C03625=1058.600,403.562,-118.922,174.891,38.797,157.435
C03626=1058.591,403.315,-118.879,174.884,38.789,157.432
C03627=1058.583,403.069,-118.835,174.877,38.781,157.430
C03628=1058.575,402.823,-118.792,174.870,38.773,157.428
C03629=1058.566,402.577,-118.749,174.863,38.765,157.426
C03630=1058.556,402.249,-118.691,174.854,38.754,157.423
C03631=1058.545,401.921,-118.634,174.845,38.744,157.420
C03632=1058.534,401.593,-118.577,174.836,38.733,157.417
C03633=1058.523,401.265,-118.519,174.828,38.723,157.414
C03634=1058.515,401.019,-118.477,174.821,38.715,157.412
C03635=1058.506,400.773,-118.434,174.814,38.707,157.410
C03636=1058.498,400.527,-118.391,174.807,38.699,157.408
C03637=1058.489,400.280,-118.348,174.800,38.691,157.406
C03638=1058.483,400.034,-118.305,174.794,38.684,157.404
C03639=1058.474,399.788,-118.262,174.787,38.676,157.402
C03640=1058.466,399.542,-118.219,174.781,38.668,157.400
C03641=1058.457,399.295,-118.177,174.774,38.660,157.398
C03642=1058.449,399.050,-118.134,174.768,38.652,157.395
C03643=1058.441,398.803,-118.092,174.761,38.644,157.393
C03644=1058.433,398.557,-118.049,174.754,38.637,157.391
C03645=1058.426,398.311,-118.006,174.748,38.629,157.389
C03646=1058.417,398.065,-117.963,174.742,38.622,157.387
C03647=1058.409,397.818,-117.921,174.735,38.614,157.385
C03648=1058.401,397.573,-117.878,174.729,38.606,157.383
C03649=1058.393,397.326,-117.836,174.722,38.599,157.381
C03650=1058.385,397.080,-117.794,174.716,38.591,157.379
C03651=1058.377,396.834,-117.751,174.710,38.583,157.377
C03652=1058.369,396.588,-117.709,174.703,38.576,157.375
C03653=1058.361,396.342,-117.667,174.696,38.568,157.373
C03654=1058.353,396.095,-117.624,174.691,38.561,157.371
C03655=1058.345,395.848,-117.582,174.684,38.554,157.369
C03656=1058.337,395.603,-117.539,174.677,38.546,157.367
C03657=1058.329,395.357,-117.497,174.672,38.539,157.365
C03658=1058.320,395.111,-117.456,174.665,38.531,157.363
C03659=1058.313,394.865,-117.414,174.659,38.524,157.361
C03660=1058.305,394.618,-117.371,174.652,38.516,157.359
C03661=1058.297,394.372,-117.330,174.647,38.509,157.357
C03662=1058.289,394.125,-117.287,174.640,38.502,157.355
C03663=1058.281,393.879,-117.245,174.633,38.494,157.353
C03664=1058.273,393.633,-117.203,174.628,38.487,157.351
C03665=1058.265,393.387,-117.161,174.621,38.479,157.349
C03666=1058.258,393.141,-117.119,174.615,38.472,157.348
C03667=1058.249,392.894,-117.078,174.609,38.465,157.346
C03668=1058.242,392.648,-117.036,174.603,38.458,157.344
C03669=1058.234,392.402,-116.994,174.597,38.451,157.342
C03670=1058.226,392.155,-116.952,174.591,38.444,157.340
C03671=1058.218,391.909,-116.911,174.584,38.436,157.338
C03672=1058.210,391.663,-116.869,174.579,38.429,157.336
C03673=1058.202,391.416,-116.827,174.572,38.422,157.334
C03674=1058.194,391.170,-116.786,174.566,38.415,157.332
C03675=1058.186,390.924,-116.744,174.560,38.408,157.330
C03676=1058.179,390.677,-116.703,174.554,38.400,157.328
C03677=1058.171,390.431,-116.661,174.548,38.393,157.327
C03678=1058.163,390.184,-116.620,174.542,38.386,157.325
C03679=1058.155,389.938,-116.578,174.537,38.379,157.323
C03680=1058.147,389.692,-116.538,174.530,38.372,157.321
C03681=1058.140,389.446,-116.496,174.525,38.365,157.319
C03682=1058.131,389.199,-116.455,174.518,38.359,157.318
C03683=1058.124,388.953,-116.413,174.512,38.352,157.316
C03684=1058.116,388.706,-116.373,174.506,38.345,157.314
C03685=1058.108,388.460,-116.331,174.500,38.338,157.312
C03686=1058.098,388.150,-116.280,174.493,38.329,157.310
C03687=1058.088,387.839,-116.228,174.486,38.320,157.308
C03688=1058.079,387.528,-116.176,174.478,38.312,157.305
C03689=1058.069,387.217,-116.124,174.471,38.303,157.303
C03690=1058.061,386.971,-116.082,174.464,38.296,157.301
C03691=1058.053,386.725,-116.042,174.459,38.289,157.299
C03692=1058.045,386.479,-116.001,174.453,38.283,157.298
C03693=1058.038,386.232,-115.960,174.447,38.276,157.296
C03694=1058.030,385.986,-115.919,174.441,38.269,157.294
C03695=1058.022,385.739,-115.878,174.436,38.262,157.292
C03696=1058.014,385.492,-115.837,174.431,38.255,157.291
C03697=1058.007,385.246,-115.798,174.424,38.249,157.289
C03698=1057.999,385.000,-115.756,174.419,38.242,157.287
C03699=1057.991,384.753,-115.716,174.413,38.235,157.285
C03700=1057.984,384.507,-115.674,174.407,38.229,157.284
C03701=1057.976,384.260,-115.634,174.401,38.222,157.282
C03702=1057.968,384.014,-115.593,174.396,38.215,157.280
C03703=1057.961,383.767,-115.553,174.391,38.209,157.279
C03704=1057.953,383.521,-115.512,174.384,38.202,157.277
C03705=1057.946,383.274,-115.471,174.379,38.196,157.275
C03706=1057.938,383.027,-115.431,174.373,38.189,157.273
C03707=1057.930,382.781,-115.390,174.368,38.183,157.272
C03708=1057.923,382.535,-115.349,174.362,38.176,157.270
C03709=1057.915,382.288,-115.309,174.356,38.169,157.268
C03710=1057.907,382.042,-115.269,174.351,38.163,157.267
C03711=1057.900,381.795,-115.228,174.345,38.156,157.265
C03712=1057.892,381.548,-115.188,174.340,38.150,157.263
C03713=1057.885,381.302,-115.148,174.334,38.143,157.262
C03714=1057.878,381.056,-115.107,174.328,38.137,157.260
C03715=1057.870,380.809,-115.067,174.323,38.130,157.258
C03716=1057.862,380.562,-115.026,174.318,38.124,157.257
C03717=1057.856,380.316,-114.986,174.312,38.117,157.255
C03718=1057.848,380.069,-114.946,174.307,38.111,157.253
C03719=1057.840,379.823,-114.906,174.301,38.105,157.252
C03720=1057.832,379.576,-114.866,174.295,38.098,157.250
C03721=1057.825,379.329,-114.826,174.290,38.092,157.248
C03722=1057.818,379.083,-114.786,174.285,38.086,157.247
C03723=1057.810,378.836,-114.746,174.279,38.079,157.245
C03724=1057.802,378.589,-114.706,174.274,38.073,157.244
C03725=1057.795,378.343,-114.666,174.269,38.067,157.242
C03726=1057.787,378.096,-114.626,174.263,38.060,157.240
C03727=1057.779,377.849,-114.586,174.257,38.054,157.239
C03728=1057.772,377.603,-114.547,174.252,38.048,157.237
C03729=1057.764,377.356,-114.507,174.247,38.042,157.236
C03730=1057.757,377.109,-114.467,174.241,38.035,157.234
C03731=1057.750,376.863,-114.427,174.236,38.029,157.233
C03732=1057.742,376.616,-114.387,174.231,38.023,157.231
C03733=1057.734,376.369,-114.348,174.226,38.017,157.229
C03734=1057.727,376.123,-114.308,174.220,38.011,157.228
C03735=1057.719,375.876,-114.268,174.215,38.004,157.226
C03736=1057.713,375.629,-114.229,174.210,37.998,157.225
C03737=1057.705,375.383,-114.189,174.205,37.992,157.223
C03738=1057.698,375.136,-114.150,174.199,37.986,157.221
C03739=1057.690,374.889,-114.110,174.194,37.980,157.220
C03740=1057.683,374.643,-114.070,174.189,37.974,157.218
C03741=1057.675,374.396,-114.031,174.184,37.968,157.217
C03742=1057.667,374.117,-113.986,174.177,37.961,157.215
C03743=1057.659,373.838,-113.942,174.171,37.954,157.213
C03744=1057.650,373.559,-113.898,174.166,37.947,157.212
C03745=1057.642,373.279,-113.853,174.159,37.940,157.210
C03746=1057.635,373.033,-113.813,174.154,37.934,157.208
C03747=1057.627,372.786,-113.773,174.149,37.928,157.207
C03748=1057.621,372.539,-113.735,174.145,37.922,157.205
C03749=1057.613,372.292,-113.695,174.139,37.916,157.204
C03750=1057.606,372.045,-113.656,174.134,37.910,157.202
C03751=1057.598,371.799,-113.617,174.129,37.905,157.201
C03752=1057.591,371.552,-113.578,174.124,37.899,157.199
C03753=1057.584,371.305,-113.539,174.119,37.893,157.198
C03754=1057.575,371.059,-113.500,174.114,37.887,157.196
C03755=1057.569,370.812,-113.461,174.108,37.881,157.195
C03756=1057.561,370.564,-113.421,174.103,37.875,157.194
C03757=1057.553,370.318,-113.383,174.098,37.869,157.192
C03758=1057.547,370.072,-113.344,174.093,37.863,157.191
C03759=1057.539,369.824,-113.304,174.088,37.858,157.189
C03760=1057.532,369.577,-113.266,174.083,37.852,157.188
C03761=1057.525,369.331,-113.227,174.078,37.846,157.186
C03762=1057.516,369.084,-113.188,174.073,37.840,157.185
C03763=1057.510,368.837,-113.149,174.067,37.834,157.183
C03764=1057.503,368.590,-113.110,174.063,37.829,157.182
C03765=1057.495,368.343,-113.072,174.058,37.823,157.180
C03766=1057.488,368.096,-113.033,174.053,37.817,157.179
C03767=1057.480,367.850,-112.995,174.048,37.811,157.178
C03768=1057.473,367.603,-112.956,174.043,37.806,157.176
C03769=1057.466,367.355,-112.917,174.038,37.800,157.175
C03770=1057.458,367.109,-112.878,174.033,37.794,157.173
C03771=1057.452,366.862,-112.840,174.029,37.789,157.172
C03772=1057.444,366.616,-112.801,174.023,37.783,157.170
C03773=1057.437,366.369,-112.763,174.018,37.777,157.169
C03774=1057.430,366.122,-112.724,174.013,37.772,157.168
C03775=1057.423,365.874,-112.686,174.008,37.766,157.166
C03776=1057.416,365.627,-112.647,174.003,37.760,157.165
C03777=1057.408,365.381,-112.609,173.999,37.755,157.163
C03778=1057.401,365.134,-112.570,173.994,37.749,157.162
C03779=1057.394,364.887,-112.532,173.989,37.743,157.161
C03780=1057.387,364.640,-112.494,173.984,37.738,157.159
C03781=1057.381,364.393,-112.455,173.979,37.732,157.158
C03782=1057.373,364.147,-112.416,173.975,37.727,157.157
C03783=1057.366,363.900,-112.378,173.970,37.721,157.155
C03784=1057.359,363.653,-112.340,173.965,37.715,157.154
C03785=1057.351,363.406,-112.301,173.960,37.710,157.152
C03786=1057.344,363.158,-112.263,173.956,37.704,157.151
C03787=1057.337,362.912,-112.225,173.951,37.699,157.150
C03788=1057.330,362.664,-112.188,173.946,37.694,157.148
C03789=1057.323,362.418,-112.149,173.941,37.688,157.147
C03790=1057.315,362.170,-112.111,173.937,37.683,157.146
C03791=1057.308,361.924,-112.073,173.932,37.677,157.144
C03792=1057.301,361.677,-112.035,173.926,37.672,157.143
C03793=1057.294,361.430,-111.997,173.921,37.666,157.142
C03794=1057.287,361.183,-111.959,173.917,37.661,157.140
C03795=1057.279,360.936,-111.922,173.912,37.655,157.139
C03796=1057.273,360.689,-111.883,173.907,37.650,157.138
C03797=1057.265,360.442,-111.845,173.902,37.645,157.136
C03798=1057.257,360.181,-111.806,173.898,37.639,157.135
C03799=1057.250,359.921,-111.765,173.893,37.633,157.133
C03800=1057.242,359.660,-111.726,173.888,37.627,157.132
C03801=1057.235,359.399,-111.686,173.883,37.622,157.131
C03802=1057.228,359.152,-111.648,173.878,37.616,157.129
C03803=1057.220,358.905,-111.610,173.873,37.611,157.128
C03804=1057.214,358.658,-111.572,173.869,37.606,157.127
C03805=1057.207,358.411,-111.534,173.864,37.600,157.125
C03806=1057.200,358.164,-111.497,173.860,37.595,157.124
C03807=1057.193,357.917,-111.459,173.855,37.590,157.123
C03808=1057.185,357.670,-111.422,173.851,37.585,157.122
C03809=1057.178,357.423,-111.384,173.847,37.579,157.120
C03810=1057.171,357.176,-111.347,173.842,37.574,157.119
C03811=1057.164,356.928,-111.309,173.837,37.569,157.118
C03812=1057.157,356.682,-111.272,173.833,37.564,157.117
C03813=1057.151,356.435,-111.234,173.828,37.558,157.115
C03814=1057.143,356.187,-111.197,173.823,37.553,157.114
C03815=1057.136,355.940,-111.159,173.819,37.548,157.113
C03816=1057.129,355.693,-111.121,173.814,37.543,157.111
C03817=1057.122,355.445,-111.085,173.809,37.538,157.110
C03818=1057.115,355.199,-111.047,173.805,37.533,157.109
C03819=1057.108,354.952,-111.010,173.800,37.527,157.108
C03820=1057.101,354.705,-110.972,173.796,37.522,157.106
C03821=1057.094,354.458,-110.935,173.791,37.517,157.105
C03822=1057.087,354.210,-110.898,173.786,37.512,157.104
C03823=1057.080,353.963,-110.861,173.782,37.507,157.103
C03824=1057.073,353.716,-110.823,173.778,37.502,157.101
C03825=1057.066,353.468,-110.787,173.774,37.497,157.100
C03826=1057.059,353.222,-110.749,173.769,37.492,157.099
C03827=1057.052,352.975,-110.712,173.765,37.486,157.098
C03828=1057.045,352.727,-110.675,173.760,37.481,157.096
C03829=1057.038,352.481,-110.638,173.756,37.476,157.095
C03830=1057.031,352.233,-110.601,173.751,37.471,157.094
C03831=1057.023,351.986,-110.564,173.746,37.466,157.093
C03832=1057.017,351.740,-110.527,173.742,37.461,157.092
C03833=1057.010,351.492,-110.490,173.738,37.456,157.090
C03834=1057.003,351.245,-110.453,173.734,37.451,157.089
C03835=1056.996,350.998,-110.416,173.729,37.446,157.088
C03836=1056.989,350.750,-110.379,173.725,37.441,157.087
C03837=1056.983,350.504,-110.342,173.720,37.436,157.086
C03838=1056.975,350.256,-110.306,173.716,37.431,157.084
C03839=1056.968,350.008,-110.269,173.711,37.426,157.083
C03840=1056.961,349.762,-110.232,173.707,37.421,157.082
C03841=1056.954,349.514,-110.195,173.703,37.416,157.081
C03842=1056.947,349.267,-110.159,173.699,37.411,157.080
C03843=1056.940,349.020,-110.122,173.694,37.406,157.078
C03844=1056.933,348.772,-110.085,173.690,37.401,157.077
C03845=1056.926,348.526,-110.049,173.685,37.397,157.076
C03846=1056.919,348.278,-110.012,173.681,37.392,157.075
C03847=1056.913,348.032,-109.975,173.676,37.387,157.074
C03848=1056.906,347.784,-109.938,173.673,37.382,157.072
C03849=1056.899,347.537,-109.903,173.668,37.377,157.071
C03850=1056.892,347.289,-109.866,173.664,37.372,157.070
C03851=1056.885,347.042,-109.829,173.660,37.367,157.069
C03852=1056.878,346.795,-109.793,173.655,37.362,157.068
C03853=1056.871,346.548,-109.757,173.651,37.358,157.067
C03854=1056.864,346.292,-109.719,173.647,37.353,157.066
C03855=1056.857,346.035,-109.681,173.643,37.348,157.064
C03856=1056.850,345.780,-109.643,173.638,37.343,157.063
C03857=1056.843,345.524,-109.605,173.633,37.338,157.062
C03858=1056.836,345.277,-109.570,173.629,37.333,157.061
C03859=1056.829,345.029,-109.533,173.625,37.327,157.060
C03860=1056.823,344.782,-109.497,173.621,37.323,157.058
C03861=1056.815,344.535,-109.461,173.617,37.318,157.057
C03862=1056.809,344.288,-109.424,173.612,37.314,157.056
C03863=1056.802,344.041,-109.388,173.608,37.308,157.055
C03864=1056.795,343.793,-109.352,173.604,37.304,157.054
C03865=1056.788,343.546,-109.315,173.600,37.299,157.053
C03866=1056.781,343.298,-109.280,173.596,37.295,157.052
C03867=1056.775,343.051,-109.243,173.592,37.289,157.050
C03868=1056.767,342.804,-109.207,173.587,37.285,157.049
C03869=1056.761,342.557,-109.171,173.583,37.280,157.048
C03870=1056.754,342.309,-109.135,173.579,37.275,157.047
C03871=1056.747,342.062,-109.100,173.575,37.271,157.046
C03872=1056.740,341.815,-109.063,173.571,37.266,157.045
C03873=1056.733,341.567,-109.028,173.566,37.261,157.044
C03874=1056.726,341.321,-108.992,173.562,37.257,157.043
C03875=1056.719,341.072,-108.956,173.559,37.252,157.042
C03876=1056.712,340.826,-108.920,173.554,37.247,157.040
C03877=1056.706,340.578,-108.883,173.550,37.243,157.039
C03878=1056.698,340.330,-108.848,173.546,37.238,157.038
C03879=1056.691,340.084,-108.812,173.542,37.233,157.037
C03880=1056.685,339.836,-108.776,173.538,37.229,157.036
C03881=1056.678,339.589,-108.740,173.534,37.224,157.035
C03882=1056.671,339.341,-108.705,173.529,37.219,157.034
C03883=1056.665,339.093,-108.669,173.526,37.215,157.033
C03884=1056.658,338.847,-108.633,173.522,37.210,157.032
C03885=1056.651,338.599,-108.598,173.517,37.206,157.031
C03886=1056.644,338.352,-108.561,173.513,37.201,157.030
C03887=1056.637,338.104,-108.526,173.510,37.197,157.029
C03888=1056.631,337.857,-108.491,173.506,37.192,157.027
C03889=1056.624,337.610,-108.455,173.501,37.187,157.026
C03890=1056.617,337.362,-108.420,173.497,37.183,157.025
C03891=1056.611,337.115,-108.384,173.494,37.178,157.024
C03892=1056.604,336.868,-108.349,173.489,37.174,157.023
C03893=1056.597,336.620,-108.312,173.485,37.169,157.022
C03894=1056.590,336.373,-108.277,173.481,37.165,157.021
C03895=1056.583,336.125,-108.242,173.478,37.160,157.020
C03896=1056.577,335.878,-108.207,173.473,37.156,157.019
C03897=1056.570,335.631,-108.172,173.469,37.151,157.018
C03898=1056.563,335.384,-108.136,173.465,37.147,157.017
C03899=1056.555,335.136,-108.101,173.462,37.142,157.016
C03900=1056.549,334.888,-108.065,173.457,37.138,157.015
C03901=1056.543,334.641,-108.030,173.453,37.133,157.014
C03902=1056.536,334.393,-107.995,173.450,37.129,157.013
C03903=1056.529,334.146,-107.959,173.446,37.124,157.011
C03904=1056.522,333.899,-107.924,173.442,37.120,157.010
C03905=1056.516,333.651,-107.889,173.437,37.115,157.009
C03906=1056.509,333.404,-107.854,173.434,37.111,157.008
C03907=1056.502,333.156,-107.819,173.430,37.107,157.007
C03908=1056.495,332.909,-107.784,173.426,37.102,157.006
C03909=1056.489,332.662,-107.749,173.422,37.098,157.005
C03910=1056.482,332.401,-107.712,173.418,37.093,157.004
C03911=1056.475,332.141,-107.675,173.414,37.088,157.003
C03912=1056.468,331.881,-107.638,173.409,37.084,157.002
C03913=1056.461,331.621,-107.601,173.406,37.079,157.001
C03914=1056.454,331.373,-107.566,173.402,37.075,157.000
C03915=1056.447,331.126,-107.531,173.398,37.070,156.999
C03916=1056.441,330.878,-107.496,173.395,37.066,156.998
C03917=1056.434,330.630,-107.461,173.390,37.062,156.997
C03918=1056.427,330.383,-107.426,173.386,37.057,156.996
C03919=1056.420,330.136,-107.391,173.383,37.053,156.995
C03920=1056.413,329.888,-107.357,173.379,37.049,156.994
C03921=1056.406,329.641,-107.322,173.375,37.044,156.993
C03922=1056.400,329.393,-107.287,173.372,37.040,156.992
C03923=1056.392,329.146,-107.253,173.367,37.036,156.991
C03924=1056.386,328.898,-107.218,173.363,37.032,156.990
C03925=1056.379,328.650,-107.183,173.360,37.027,156.989
C03926=1056.372,328.403,-107.149,173.356,37.023,156.988
C03927=1056.365,328.155,-107.114,173.352,37.019,156.987
C03928=1056.359,327.909,-107.080,173.349,37.015,156.986
C03929=1056.352,327.661,-107.046,173.344,37.010,156.985
C03930=1056.345,327.414,-107.011,173.340,37.006,156.984
C03931=1056.339,327.166,-106.976,173.337,37.002,156.983
C03932=1056.331,326.919,-106.942,173.333,36.998,156.982
C03933=1056.325,326.671,-106.907,173.329,36.993,156.981
C03934=1056.318,326.423,-106.872,173.326,36.989,156.980
C03935=1056.311,326.176,-106.838,173.322,36.985,156.979
C03936=1056.304,325.928,-106.804,173.318,36.981,156.978
C03937=1056.297,325.681,-106.769,173.315,36.977,156.977
C03938=1056.291,325.433,-106.735,173.310,36.972,156.976
C03939=1056.284,325.185,-106.701,173.307,36.968,156.975
C03940=1056.277,324.938,-106.666,173.303,36.964,156.974
C03941=1056.270,324.690,-106.632,173.299,36.960,156.973
C03942=1056.264,324.442,-106.597,173.296,36.956,156.972
C03943=1056.257,324.196,-106.563,173.292,36.951,156.971
C03944=1056.251,323.948,-106.529,173.288,36.947,156.970
C03945=1056.243,323.700,-106.495,173.285,36.943,156.969
C03946=1056.237,323.452,-106.461,173.281,36.939,156.968
C03947=1056.231,323.206,-106.426,173.277,36.935,156.968
C03948=1056.224,322.958,-106.392,173.274,36.931,156.967
C03949=1056.217,322.710,-106.358,173.270,36.926,156.966
C03950=1056.210,322.462,-106.324,173.267,36.922,156.965
C03951=1056.204,322.215,-106.290,173.263,36.918,156.964
C03952=1056.197,321.967,-106.256,173.259,36.913,156.963
C03953=1056.190,321.719,-106.221,173.256,36.909,156.962
C03954=1056.184,321.472,-106.187,173.252,36.906,156.961
C03955=1056.177,321.224,-106.154,173.248,36.901,156.960
C03956=1056.170,320.977,-106.118,173.244,36.897,156.959
C03957=1056.164,320.730,-106.085,173.240,36.893,156.958
C03958=1056.157,320.482,-106.051,173.237,36.889,156.957
C03959=1056.150,320.234,-106.017,173.233,36.884,156.956
C03960=1056.144,319.987,-105.983,173.229,36.880,156.955
C03961=1056.137,319.739,-105.949,173.226,36.876,156.954
C03962=1056.131,319.491,-105.914,173.223,36.872,156.953
C03963=1056.125,319.243,-105.881,173.219,36.868,156.952
C03964=1056.118,318.996,-105.847,173.216,36.864,156.951
C03965=1056.112,318.749,-105.813,173.212,36.860,156.950
C03966=1056.104,318.483,-105.777,173.208,36.855,156.949
C03967=1056.098,318.218,-105.741,173.204,36.851,156.948
C03968=1056.090,317.952,-105.704,173.200,36.847,156.947
C03969=1056.084,317.686,-105.668,173.197,36.842,156.946
C03970=1056.077,317.439,-105.634,173.193,36.838,156.946
C03971=1056.071,317.191,-105.600,173.190,36.834,156.945
C03972=1056.064,316.944,-105.566,173.186,36.830,156.944
C03973=1056.058,316.696,-105.532,173.182,36.826,156.943
C03974=1056.051,316.448,-105.499,173.179,36.822,156.942
C03975=1056.045,316.201,-105.465,173.175,36.818,156.941
C03976=1056.038,315.953,-105.431,173.172,36.814,156.940
C03977=1056.032,315.706,-105.397,173.168,36.810,156.939
C03978=1056.026,315.458,-105.365,173.164,36.806,156.938
C03979=1056.019,315.210,-105.330,173.162,36.801,156.937
C03980=1056.013,314.963,-105.297,173.158,36.797,156.936
C03981=1056.007,314.715,-105.263,173.155,36.793,156.935
C03982=1056.000,314.468,-105.229,173.151,36.789,156.934
C03983=1055.994,314.220,-105.195,173.147,36.785,156.933
C03984=1055.987,313.972,-105.162,173.144,36.781,156.933
C03985=1055.981,313.725,-105.129,173.140,36.777,156.932
C03986=1055.975,313.477,-105.095,173.137,36.773,156.931
C03987=1055.968,313.230,-105.062,173.133,36.769,156.930
C03988=1055.961,312.981,-105.029,173.130,36.765,156.929
C03989=1055.954,312.734,-104.995,173.126,36.761,156.928
C03990=1055.948,312.486,-104.962,173.123,36.757,156.927
C03991=1055.941,312.239,-104.929,173.120,36.753,156.926
C03992=1055.934,311.991,-104.895,173.116,36.749,156.925
C03993=1055.928,311.743,-104.863,173.113,36.745,156.925
C03994=1055.921,311.495,-104.830,173.109,36.741,156.924
C03995=1055.914,311.248,-104.796,173.106,36.737,156.923
C03996=1055.908,311.000,-104.763,173.102,36.734,156.922
C03997=1055.901,310.752,-104.730,173.099,36.730,156.921
C03998=1055.894,310.505,-104.697,173.095,36.726,156.920
C03999=1055.887,310.257,-104.664,173.091,36.722,156.919
C04000=1055.881,310.010,-104.632,173.089,36.718,156.918
C04001=1055.874,309.762,-104.599,173.085,36.714,156.918
C04002=1055.867,309.514,-104.565,173.082,36.710,156.917
C04003=1055.861,309.267,-104.532,173.078,36.706,156.916
C04004=1055.854,309.019,-104.500,173.075,36.702,156.915
C04005=1055.848,308.771,-104.466,173.071,36.699,156.914
C04006=1055.841,308.523,-104.434,173.068,36.695,156.913
C04007=1055.835,308.276,-104.401,173.065,36.691,156.912
C04008=1055.828,308.028,-104.367,173.062,36.687,156.911
C04009=1055.821,307.781,-104.335,173.058,36.683,156.911
C04010=1055.814,307.533,-104.302,173.055,36.679,156.910
C04011=1055.808,307.285,-104.269,173.051,36.675,156.909
C04012=1055.801,307.037,-104.236,173.047,36.672,156.908
C04013=1055.795,306.790,-104.204,173.044,36.668,156.907
C04014=1055.789,306.542,-104.171,173.041,36.664,156.906
C04015=1055.782,306.294,-104.138,173.038,36.660,156.905
C04016=1055.775,306.046,-104.105,173.034,36.656,156.905
C04017=1055.768,305.799,-104.073,173.031,36.652,156.904
C04018=1055.762,305.551,-104.040,173.027,36.649,156.903
C04019=1055.755,305.303,-104.007,173.025,36.645,156.902
C04020=1055.749,305.055,-103.974,173.021,36.641,156.901
C04021=1055.743,304.808,-103.942,173.018,36.637,156.900
C04022=1055.736,304.546,-103.907,173.014,36.633,156.899
C04023=1055.730,304.285,-103.873,173.011,36.629,156.898
C04024=1055.722,304.024,-103.838,173.007,36.625,156.897
C04025=1055.715,303.762,-103.804,173.003,36.621,156.897
C04026=1055.708,303.515,-103.771,173.000,36.617,156.896
C04027=1055.702,303.267,-103.739,172.997,36.613,156.895
C04028=1055.696,303.020,-103.706,172.994,36.609,156.894
C04029=1055.690,302.772,-103.674,172.990,36.606,156.893
C04030=1055.684,302.524,-103.641,172.987,36.602,156.892
C04031=1055.677,302.276,-103.609,172.984,36.598,156.892
C04032=1055.670,302.029,-103.576,172.981,36.594,156.891
C04033=1055.664,301.780,-103.544,172.977,36.590,156.890
C04034=1055.657,301.533,-103.511,172.974,36.587,156.889
C04035=1055.651,301.285,-103.478,172.971,36.583,156.888
C04036=1055.645,301.037,-103.446,172.968,36.579,156.887
C04037=1055.638,300.790,-103.414,172.964,36.575,156.886
C04038=1055.632,300.542,-103.382,172.962,36.571,156.886
C04039=1055.625,300.294,-103.349,172.958,36.568,156.885
C04040=1055.619,300.046,-103.317,172.955,36.563,156.884
C04041=1055.613,299.799,-103.284,172.951,36.559,156.883
C04042=1055.607,299.574,-103.255,172.949,36.556,156.882
C04043=1055.601,299.351,-103.226,172.945,36.552,156.881
C04044=1055.595,299.126,-103.197,172.943,36.549,156.881
C04045=1055.590,298.903,-103.168,172.940,36.546,156.880
C04046=1055.584,298.678,-103.139,172.937,36.542,156.879
C04047=1055.579,298.455,-103.110,172.934,36.539,156.879
C04048=1055.573,298.230,-103.080,172.931,36.536,156.878
C04049=1055.568,298.007,-103.050,172.929,36.532,156.877
C04050=1055.562,297.759,-103.018,172.925,36.528,156.876
C04051=1055.555,297.511,-102.987,172.923,36.524,156.875
C04052=1055.549,297.263,-102.954,172.919,36.521,156.874
C04053=1055.543,297.015,-102.922,172.916,36.517,156.874
C04054=1055.536,296.768,-102.889,172.913,36.513,156.873
C04055=1055.530,296.520,-102.858,172.910,36.509,156.872
C04056=1055.523,296.272,-102.825,172.906,36.506,156.871
C04057=1055.517,296.024,-102.794,172.904,36.502,156.870
C04058=1055.511,295.776,-102.762,172.900,36.498,156.869
C04059=1055.504,295.529,-102.730,172.897,36.495,156.869
C04060=1055.498,295.280,-102.698,172.894,36.491,156.868
C04061=1055.491,295.033,-102.666,172.891,36.487,156.867
C04062=1055.485,294.784,-102.634,172.887,36.483,156.866
C04063=1055.478,294.537,-102.602,172.885,36.479,156.865
C04064=1055.471,294.289,-102.571,172.881,36.476,156.865
C04065=1055.465,294.041,-102.539,172.878,36.472,156.864
C04066=1055.458,293.793,-102.507,172.875,36.468,156.863
C04067=1055.452,293.545,-102.474,172.872,36.465,156.862
C04068=1055.445,293.298,-102.443,172.868,36.461,156.861
C04069=1055.439,293.050,-102.412,172.866,36.457,156.861
C04070=1055.433,292.802,-102.380,172.862,36.454,156.860
C04071=1055.427,292.554,-102.348,172.859,36.450,156.859
C04072=1055.420,292.306,-102.317,172.856,36.446,156.858
C04073=1055.414,292.058,-102.285,172.853,36.443,156.857
C04074=1055.407,291.810,-102.254,172.850,36.439,156.856
C04075=1055.400,291.562,-102.222,172.847,36.435,156.856
C04076=1055.394,291.314,-102.190,172.844,36.432,156.855
C04077=1055.387,291.067,-102.158,172.841,36.428,156.854
C04078=1055.380,290.774,-102.121,172.838,36.424,156.853
C04079=1055.373,290.481,-102.084,172.834,36.419,156.852
C04080=1055.365,290.188,-102.047,172.830,36.415,156.851
C04081=1055.357,289.895,-102.009,172.826,36.410,156.850
C04082=1055.351,289.646,-101.977,172.823,36.407,156.850
C04083=1055.345,289.399,-101.946,172.820,36.403,156.849
C04084=1055.338,289.151,-101.915,172.817,36.400,156.848
C04085=1055.332,288.903,-101.883,172.814,36.396,156.847
C04086=1055.326,288.654,-101.852,172.812,36.392,156.846
C04087=1055.319,288.407,-101.821,172.808,36.389,156.846
C04088=1055.313,288.159,-101.790,172.805,36.385,156.845
C04089=1055.306,287.911,-101.758,172.802,36.381,156.844
C04090=1055.300,287.664,-101.727,172.799,36.378,156.843
C04091=1055.293,287.416,-101.695,172.796,36.374,156.842
C04092=1055.287,287.167,-101.664,172.793,36.371,156.842
C04093=1055.281,286.920,-101.633,172.790,36.367,156.841
C04094=1055.274,286.672,-101.602,172.787,36.363,156.840
C04095=1055.268,286.424,-101.570,172.783,36.360,156.839
C04096=1055.261,286.175,-101.539,172.781,36.356,156.839
C04097=1055.254,285.927,-101.508,172.778,36.353,156.838
C04098=1055.248,285.680,-101.477,172.775,36.349,156.837
C04099=1055.242,285.432,-101.446,172.772,36.346,156.836
C04100=1055.235,285.184,-101.415,172.769,36.342,156.835
C04101=1055.228,284.936,-101.383,172.766,36.338,156.835
C04102=1055.223,284.688,-101.353,172.763,36.335,156.834
C04103=1055.216,284.440,-101.322,172.760,36.331,156.833
C04104=1055.209,284.192,-101.291,172.757,36.328,156.832
C04105=1055.203,283.944,-101.260,172.754,36.324,156.832
C04106=1055.197,283.697,-101.228,172.752,36.320,156.831
C04107=1055.190,283.448,-101.198,172.748,36.316,156.830
C04108=1055.184,283.201,-101.167,172.746,36.313,156.829
C04109=1055.178,282.952,-101.136,172.742,36.309,156.828
C04110=1055.171,282.704,-101.104,172.740,36.306,156.828
C04111=1055.165,282.457,-101.074,172.736,36.302,156.827
C04112=1055.158,282.209,-101.043,172.734,36.299,156.826
C04113=1055.152,281.960,-101.012,172.730,36.295,156.825
C04114=1055.146,281.713,-100.981,172.728,36.291,156.824
C04115=1055.139,281.464,-100.950,172.725,36.288,156.824
C04116=1055.133,281.216,-100.919,172.722,36.284,156.823
C04117=1055.127,280.969,-100.888,172.719,36.281,156.822
C04118=1055.120,280.720,-100.858,172.716,36.277,156.821
C04119=1055.114,280.473,-100.827,172.713,36.273,156.821
C04120=1055.108,280.224,-100.796,172.710,36.270,156.820
C04121=1055.102,279.976,-100.765,172.707,36.266,156.819
C04122=1055.095,279.729,-100.734,172.705,36.263,156.818
C04123=1055.089,279.480,-100.703,172.701,36.259,156.818
C04124=1055.083,279.232,-100.673,172.699,36.256,156.817
C04125=1055.076,278.984,-100.642,172.695,36.252,156.816
C04126=1055.069,278.736,-100.611,172.693,36.249,156.815
C04127=1055.063,278.488,-100.581,172.691,36.245,156.815
C04128=1055.057,278.240,-100.550,172.687,36.242,156.814
C04129=1055.051,277.992,-100.520,172.685,36.238,156.813
C04130=1055.044,277.751,-100.490,172.681,36.234,156.812
C04131=1055.038,277.510,-100.460,172.679,36.231,156.812
C04132=1055.032,277.269,-100.431,172.675,36.227,156.811
C04133=1055.026,277.027,-100.400,172.673,36.224,156.810
C04134=1055.020,276.786,-100.371,172.671,36.220,156.809
C04135=1055.013,276.545,-100.342,172.667,36.217,156.809
C04136=1055.007,276.304,-100.312,172.665,36.213,156.808
C04137=1055.001,276.062,-100.282,172.662,36.210,156.807
C04138=1054.994,275.815,-100.252,172.659,36.207,156.806
C04139=1054.988,275.566,-100.221,172.657,36.203,156.806
C04140=1054.982,275.318,-100.191,172.653,36.199,156.805
C04141=1054.975,275.070,-100.161,172.651,36.196,156.804
C04142=1054.969,274.822,-100.130,172.648,36.192,156.803
C04143=1054.963,274.574,-100.100,172.645,36.189,156.803
C04144=1054.956,274.326,-100.070,172.642,36.185,156.802
C04145=1054.950,274.078,-100.039,172.639,36.182,156.801
C04146=1054.944,273.830,-100.009,172.637,36.178,156.800
C04147=1054.937,273.582,-99.979,172.634,36.175,156.800
C04148=1054.931,273.334,-99.948,172.631,36.171,156.799
C04149=1054.925,273.086,-99.918,172.628,36.168,156.798
C04150=1054.918,272.838,-99.888,172.626,36.164,156.797
C04151=1054.912,272.590,-99.858,172.623,36.161,156.797
C04152=1054.906,272.342,-99.827,172.620,36.157,156.796
C04153=1054.900,272.093,-99.798,172.617,36.153,156.795
C04154=1054.893,271.845,-99.767,172.614,36.150,156.794
C04155=1054.887,271.597,-99.737,172.612,36.146,156.794
C04156=1054.880,271.349,-99.707,172.609,36.143,156.793
C04157=1054.874,271.101,-99.677,172.606,36.139,156.792
C04158=1054.868,270.854,-99.647,172.604,36.136,156.791
C04159=1054.861,270.605,-99.617,172.600,36.133,156.791
C04160=1054.855,270.357,-99.587,172.598,36.129,156.790
C04161=1054.848,270.109,-99.557,172.595,36.126,156.789
C04162=1054.842,269.861,-99.526,172.592,36.122,156.788
C04163=1054.835,269.612,-99.497,172.590,36.119,156.788
C04164=1054.830,269.364,-99.467,172.586,36.115,156.787
C04165=1054.823,269.117,-99.437,172.584,36.112,156.786
C04166=1054.817,268.868,-99.407,172.582,36.108,156.785
C04167=1054.810,268.620,-99.377,172.578,36.105,156.785
C04168=1054.805,268.372,-99.347,172.576,36.101,156.784
C04169=1054.798,268.123,-99.317,172.573,36.098,156.783
C04170=1054.791,267.876,-99.287,172.570,36.094,156.782
C04171=1054.785,267.627,-99.257,172.568,36.090,156.782
C04172=1054.778,267.379,-99.228,172.565,36.087,156.781
C04173=1054.772,267.132,-99.198,172.562,36.083,156.780
C04174=1054.766,266.883,-99.168,172.559,36.080,156.779
C04175=1054.759,266.635,-99.138,172.557,36.076,156.779
C04176=1054.753,266.387,-99.109,172.555,36.073,156.778
C04177=1054.747,266.138,-99.078,172.551,36.070,156.777
C04178=1054.740,265.890,-99.049,172.549,36.066,156.777
C04179=1054.734,265.643,-99.020,172.546,36.063,156.776
C04180=1054.728,265.394,-98.990,172.543,36.059,156.775
C04181=1054.721,265.146,-98.960,172.541,36.056,156.774
C04182=1054.715,264.898,-98.931,172.538,36.052,156.774
C04183=1054.709,264.650,-98.901,172.535,36.049,156.773
C04184=1054.702,264.401,-98.871,172.533,36.045,156.772
C04185=1054.696,264.154,-98.841,172.530,36.041,156.771
C04186=1054.690,263.915,-98.813,172.528,36.039,156.771
C04187=1054.683,263.675,-98.784,172.525,36.035,156.770
C04188=1054.678,263.436,-98.756,172.522,36.031,156.769
C04189=1054.672,263.197,-98.728,172.520,36.028,156.768
C04190=1054.665,262.958,-98.699,172.517,36.025,156.768
C04191=1054.659,262.719,-98.670,172.515,36.021,156.767
C04192=1054.653,262.480,-98.642,172.513,36.018,156.766
C04193=1054.647,262.240,-98.613,172.509,36.015,156.766
C04194=1054.641,261.992,-98.584,172.507,36.011,156.765
C04195=1054.635,261.744,-98.555,172.504,36.008,156.764
C04196=1054.628,261.495,-98.526,172.502,36.005,156.764
C04197=1054.620,261.248,-98.497,172.499,36.001,156.763
C04198=1054.614,260.999,-98.468,172.496,35.998,156.762
C04199=1054.607,260.751,-98.438,172.494,35.994,156.761
C04200=1054.601,260.502,-98.409,172.491,35.991,156.761
C04201=1054.595,260.254,-98.380,172.488,35.988,156.760
C04202=1054.589,260.006,-98.351,172.486,35.984,156.759
C04203=1054.581,259.758,-98.321,172.483,35.981,156.759
C04204=1054.575,259.510,-98.292,172.480,35.977,156.758
C04205=1054.569,259.262,-98.263,172.478,35.974,156.757
C04206=1054.563,259.014,-98.234,172.475,35.970,156.756
C04207=1054.556,258.765,-98.205,172.473,35.967,156.756
C04208=1054.550,258.517,-98.176,172.471,35.963,156.755
C04209=1054.543,258.268,-98.146,172.467,35.960,156.754
C04210=1054.537,258.020,-98.117,172.465,35.957,156.754
C04211=1054.531,257.772,-98.088,172.463,35.953,156.753
C04212=1054.524,257.523,-98.059,172.460,35.950,156.752
C04213=1054.518,257.275,-98.030,172.457,35.946,156.751
C04214=1054.511,257.027,-98.001,172.454,35.943,156.751
C04215=1054.505,256.779,-97.972,172.452,35.940,156.750
C04216=1054.499,256.531,-97.943,172.450,35.936,156.749
C04217=1054.492,256.283,-97.914,172.447,35.933,156.749
C04218=1054.486,256.035,-97.885,172.444,35.929,156.748
C04219=1054.479,255.786,-97.856,172.442,35.925,156.747
C04220=1054.473,255.538,-97.827,172.439,35.922,156.746
C04221=1054.466,255.290,-97.798,172.437,35.919,156.746
C04222=1054.460,255.042,-97.769,172.435,35.915,156.745
C04223=1054.454,254.794,-97.740,172.432,35.912,156.744
C04224=1054.448,254.545,-97.711,172.429,35.908,156.743
C04225=1054.442,254.297,-97.682,172.426,35.905,156.743
C04226=1054.435,254.048,-97.653,172.424,35.902,156.742
C04227=1054.429,253.800,-97.624,172.422,35.898,156.741
C04228=1054.422,253.552,-97.596,172.419,35.895,156.741
C04229=1054.415,253.304,-97.566,172.417,35.891,156.740
C04230=1054.409,253.055,-97.538,172.414,35.887,156.739
C04231=1054.403,252.807,-97.509,172.411,35.884,156.738
C04232=1054.397,252.559,-97.480,172.409,35.880,156.738
C04233=1054.391,252.311,-97.451,172.407,35.877,156.737
C04234=1054.384,252.062,-97.422,172.404,35.874,156.736
C04235=1054.378,251.814,-97.394,172.402,35.870,156.736
C04236=1054.372,251.566,-97.365,172.399,35.867,156.735
C04237=1054.365,251.318,-97.336,172.396,35.863,156.734
C04238=1054.359,251.069,-97.308,172.394,35.860,156.733
C04239=1054.353,250.821,-97.279,172.391,35.856,156.733
C04240=1054.347,250.573,-97.250,172.389,35.853,156.732
C04241=1054.340,250.325,-97.221,172.387,35.849,156.731
C04242=1054.334,250.084,-97.193,172.384,35.846,156.731
C04243=1054.329,249.844,-97.165,172.382,35.842,156.730
C04244=1054.323,249.604,-97.137,172.380,35.839,156.729
C04245=1054.316,249.364,-97.110,172.377,35.836,156.728
C04246=1054.310,249.124,-97.082,172.375,35.832,156.728
C04247=1054.304,248.884,-97.055,172.373,35.829,156.727
C04248=1054.298,248.643,-97.027,172.370,35.826,156.726
C04249=1054.293,248.404,-96.999,172.368,35.822,156.726
C04250=1054.287,248.155,-96.971,172.366,35.819,156.725
C04251=1054.281,247.907,-96.942,172.363,35.815,156.724
C04252=1054.274,247.658,-96.914,172.360,35.811,156.723
C04253=1054.268,247.410,-96.885,172.357,35.808,156.723
C04254=1054.262,247.162,-96.857,172.355,35.804,156.722
C04255=1054.255,246.913,-96.828,172.353,35.801,156.721
C04256=1054.249,246.665,-96.799,172.350,35.798,156.721
C04257=1054.244,246.417,-96.771,172.348,35.794,156.720
C04258=1054.237,246.169,-96.743,172.346,35.791,156.719
C04259=1054.231,245.921,-96.714,172.343,35.787,156.718
C04260=1054.225,245.672,-96.685,172.341,35.783,156.718
C04261=1054.218,245.424,-96.658,172.339,35.780,156.717
C04262=1054.212,245.175,-96.629,172.336,35.776,156.716
C04263=1054.205,244.927,-96.601,172.334,35.773,156.716
C04264=1054.199,244.679,-96.572,172.332,35.770,156.715
C04265=1054.193,244.430,-96.544,172.329,35.766,156.714
C04266=1054.186,244.182,-96.516,172.327,35.763,156.713
C04267=1054.181,243.934,-96.487,172.325,35.759,156.713
C04268=1054.174,243.686,-96.459,172.322,35.755,156.712
C04269=1054.168,243.437,-96.431,172.319,35.752,156.711
C04270=1054.162,243.188,-96.403,172.317,35.749,156.710
C04271=1054.155,242.940,-96.374,172.314,35.745,156.710
C04272=1054.149,242.692,-96.346,172.312,35.742,156.709
C04273=1054.143,242.444,-96.319,172.310,35.738,156.708
C04274=1054.137,242.195,-96.290,172.307,35.735,156.708
C04275=1054.130,241.947,-96.262,172.305,35.731,156.707
C04276=1054.124,241.699,-96.234,172.302,35.727,156.706
C04277=1054.118,241.450,-96.206,172.300,35.724,156.705
C04278=1054.112,241.201,-96.178,172.298,35.721,156.705
C04279=1054.105,240.953,-96.150,172.295,35.717,156.704
C04280=1054.099,240.705,-96.122,172.293,35.714,156.703
C04281=1054.093,240.457,-96.093,172.291,35.711,156.703
C04282=1054.086,240.209,-96.066,172.288,35.707,156.702
C04283=1054.079,239.960,-96.038,172.286,35.704,156.701
C04284=1054.073,239.711,-96.010,172.284,35.700,156.700
C04285=1054.067,239.463,-95.982,172.281,35.696,156.700
C04286=1054.061,239.215,-95.955,172.279,35.693,156.699
C04287=1054.055,238.967,-95.926,172.277,35.690,156.698
C04288=1054.048,238.718,-95.898,172.274,35.686,156.698
C04289=1054.041,238.470,-95.871,172.272,35.683,156.697
C04290=1054.035,238.221,-95.842,172.270,35.679,156.696
C04291=1054.029,237.973,-95.815,172.268,35.676,156.696
C04292=1054.023,237.725,-95.787,172.265,35.672,156.695
C04293=1054.017,237.476,-95.759,172.263,35.669,156.694
C04294=1054.010,237.228,-95.731,172.260,35.665,156.693
C04295=1054.003,236.979,-95.704,172.258,35.662,156.693
C04296=1053.997,236.731,-95.676,172.256,35.658,156.692
C04297=1053.991,236.483,-95.648,172.254,35.655,156.691
C04298=1053.985,236.239,-95.621,172.251,35.652,156.691
C04299=1053.979,235.997,-95.595,172.249,35.648,156.690
C04300=1053.973,235.753,-95.567,172.247,35.645,156.689
C04301=1053.966,235.510,-95.539,172.245,35.641,156.688
C04302=1053.960,235.268,-95.513,172.243,35.638,156.688
C04303=1053.954,235.024,-95.486,172.241,35.634,156.687
C04304=1053.948,234.781,-95.458,172.238,35.631,156.686
C04305=1053.941,234.537,-95.431,172.236,35.628,156.686
C04306=1053.936,234.289,-95.404,172.234,35.624,156.685
C04307=1053.929,234.040,-95.376,172.231,35.620,156.684
C04308=1053.923,233.792,-95.348,172.229,35.617,156.683
C04309=1053.917,233.544,-95.321,172.227,35.613,156.683
C04310=1053.911,233.295,-95.293,172.224,35.610,156.682
C04311=1053.904,233.046,-95.266,172.222,35.607,156.681
C04312=1053.898,232.799,-95.238,172.220,35.603,156.681
C04313=1053.892,232.550,-95.211,172.217,35.600,156.680
C04314=1053.885,232.302,-95.183,172.215,35.596,156.679
C04315=1053.879,232.053,-95.156,172.214,35.592,156.679
C04316=1053.872,231.805,-95.128,172.211,35.589,156.678
C04317=1053.866,231.556,-95.100,172.209,35.586,156.677
C04318=1053.861,231.308,-95.074,172.207,35.582,156.676
C04319=1053.854,231.059,-95.046,172.204,35.579,156.676
C04320=1053.847,230.811,-95.018,172.202,35.575,156.675
C04321=1053.842,230.563,-94.991,172.200,35.571,156.674
C04322=1053.835,230.314,-94.964,172.197,35.568,156.674
C04323=1053.829,230.066,-94.936,172.195,35.564,156.673
C04324=1053.822,229.817,-94.909,172.193,35.561,156.672
C04325=1053.816,229.569,-94.882,172.190,35.558,156.671
C04326=1053.810,229.321,-94.855,172.189,35.554,156.671
C04327=1053.803,229.072,-94.827,172.187,35.550,156.670
C04328=1053.797,228.824,-94.799,172.184,35.547,156.669
C04329=1053.791,228.575,-94.773,172.182,35.543,156.669
C04330=1053.784,228.327,-94.745,172.180,35.540,156.668
C04331=1053.778,228.079,-94.718,172.178,35.537,156.667
C04332=1053.772,227.830,-94.691,172.175,35.533,156.666
C04333=1053.765,227.581,-94.664,172.173,35.529,156.666
C04334=1053.760,227.333,-94.637,172.171,35.526,156.665
C04335=1053.753,227.084,-94.609,172.169,35.523,156.664
C04336=1053.746,226.836,-94.583,172.167,35.519,156.664
C04337=1053.740,226.588,-94.556,172.165,35.516,156.663
C04338=1053.733,226.339,-94.529,172.162,35.512,156.662
C04339=1053.727,226.091,-94.501,172.160,35.508,156.662
C04340=1053.721,225.842,-94.474,172.158,35.505,156.661
C04341=1053.715,225.593,-94.447,172.155,35.502,156.660
C04342=1053.708,225.345,-94.420,172.154,35.498,156.659
C04343=1053.702,225.097,-94.394,172.152,35.495,156.659
C04344=1053.695,224.849,-94.366,172.149,35.491,156.658
C04345=1053.689,224.599,-94.339,172.147,35.487,156.657
C04346=1053.683,224.351,-94.312,172.145,35.484,156.657
C04347=1053.676,224.103,-94.285,172.143,35.480,156.656
C04348=1053.671,223.854,-94.258,172.140,35.477,156.655
C04349=1053.664,223.605,-94.231,172.139,35.474,156.654
C04350=1053.658,223.357,-94.205,172.137,35.470,156.654
C04351=1053.651,223.109,-94.177,172.134,35.466,156.653
C04352=1053.645,222.860,-94.150,172.132,35.463,156.652
C04353=1053.639,222.611,-94.123,172.130,35.459,156.652
C04354=1053.633,222.365,-94.097,172.128,35.456,156.651
C04355=1053.626,222.118,-94.071,172.126,35.452,156.650
C04356=1053.621,221.871,-94.044,172.124,35.448,156.649
C04357=1053.614,221.624,-94.017,172.121,35.445,156.649
C04358=1053.608,221.377,-93.990,172.119,35.441,156.648
C04359=1053.602,221.130,-93.963,172.118,35.438,156.647
C04360=1053.596,220.882,-93.937,172.116,35.435,156.647
C04361=1053.589,220.636,-93.910,172.113,35.431,156.646
C04362=1053.583,220.387,-93.883,172.111,35.427,156.645
C04363=1053.576,220.139,-93.857,172.109,35.424,156.644
C04364=1053.570,219.890,-93.830,172.107,35.420,156.644
C04365=1053.563,219.642,-93.803,172.105,35.417,156.643
C04366=1053.558,219.394,-93.777,172.103,35.414,156.642
C04367=1053.551,219.145,-93.750,172.100,35.410,156.642
C04368=1053.545,218.897,-93.724,172.098,35.406,156.641
C04369=1053.538,218.648,-93.697,172.097,35.403,156.640
C04370=1053.532,218.399,-93.671,172.095,35.399,156.639
C04371=1053.525,218.150,-93.644,172.092,35.396,156.639
C04372=1053.519,217.902,-93.618,172.090,35.392,156.638
C04373=1053.512,217.653,-93.591,172.088,35.388,156.637
C04374=1053.507,217.405,-93.564,172.086,35.385,156.637
C04375=1053.500,217.157,-93.538,172.084,35.382,156.636
C04376=1053.494,216.908,-93.511,172.082,35.378,156.635
C04377=1053.487,216.660,-93.485,172.079,35.374,156.635
C04378=1053.481,216.411,-93.458,172.078,35.371,156.634
C04379=1053.474,216.163,-93.432,172.076,35.367,156.633
C04380=1053.469,215.914,-93.405,172.074,35.364,156.632
C04381=1053.462,215.666,-93.379,172.071,35.360,156.632
C04382=1053.456,215.417,-93.352,172.070,35.356,156.631
C04383=1053.450,215.169,-93.325,172.068,35.353,156.630
C04384=1053.443,214.920,-93.299,172.065,35.349,156.629
C04385=1053.437,214.671,-93.273,172.063,35.346,156.629
C04386=1053.431,214.423,-93.247,172.062,35.342,156.628
C04387=1053.425,214.174,-93.220,172.059,35.338,156.627
C04388=1053.418,213.926,-93.194,172.057,35.335,156.627
C04389=1053.412,213.678,-93.167,172.055,35.331,156.626
C04390=1053.405,213.429,-93.141,172.054,35.328,156.625
C04391=1053.399,213.181,-93.114,172.051,35.324,156.624
C04392=1053.393,212.932,-93.089,172.049,35.320,156.624
C04393=1053.387,212.683,-93.062,172.048,35.317,156.623
C04394=1053.380,212.435,-93.036,172.045,35.313,156.622
C04395=1053.374,212.186,-93.009,172.043,35.309,156.622
C04396=1053.368,211.937,-92.983,172.041,35.306,156.621
C04397=1053.362,211.689,-92.957,172.040,35.303,156.620
C04398=1053.355,211.441,-92.931,172.037,35.299,156.620
C04399=1053.348,211.192,-92.904,172.035,35.296,156.619
C04400=1053.343,210.943,-92.878,172.034,35.292,156.618
C04401=1053.336,210.695,-92.852,172.031,35.288,156.617
C04402=1053.330,210.447,-92.826,172.029,35.285,156.617
C04403=1053.324,210.197,-92.800,172.027,35.281,156.616
C04404=1053.317,209.949,-92.774,172.025,35.278,156.615
C04405=1053.311,209.701,-92.748,172.023,35.274,156.614
C04406=1053.305,209.451,-92.722,172.021,35.270,156.614
C04407=1053.298,209.203,-92.696,172.020,35.267,156.613
C04408=1053.292,208.955,-92.669,172.017,35.263,156.612
C04409=1053.286,208.706,-92.644,172.015,35.259,156.612
C04410=1053.279,208.462,-92.618,172.014,35.256,156.611
C04411=1053.273,208.218,-92.593,172.011,35.252,156.610
C04412=1053.267,207.974,-92.567,172.009,35.249,156.609
C04413=1053.261,207.729,-92.541,172.008,35.245,156.609
C04414=1053.254,207.485,-92.516,172.006,35.241,156.608
C04415=1053.249,207.240,-92.491,172.003,35.238,156.607
C04416=1053.242,206.996,-92.465,172.002,35.235,156.607
C04417=1053.236,206.752,-92.440,172.000,35.231,156.606
C04418=1053.210,205.700,-92.334,171.785,35.137,156.590
C04419=1053.204,205.451,-92.309,171.783,35.135,156.589
C04420=1053.198,205.203,-92.284,171.780,35.132,156.589
C04421=1053.192,204.954,-92.259,171.777,35.129,156.588
C04422=1053.186,204.705,-92.234,171.775,35.126,156.588
C04423=1053.180,204.456,-92.209,171.773,35.124,156.587
C04424=1053.175,204.208,-92.184,171.771,35.121,156.587
C04425=1053.168,203.959,-92.159,171.768,35.118,156.586
C04426=1053.162,203.710,-92.134,171.765,35.115,156.586
C04427=1053.156,203.462,-92.110,171.763,35.113,156.585
C04428=1053.150,203.213,-92.085,171.761,35.110,156.585
C04429=1053.144,202.964,-92.060,171.758,35.107,156.584
C04430=1053.138,202.716,-92.035,171.756,35.104,156.584
C04431=1053.133,202.467,-92.011,171.753,35.102,156.583
C04432=1053.126,202.218,-91.985,171.751,35.099,156.582
C04433=1053.121,201.970,-91.961,171.748,35.096,156.582
C04434=1053.115,201.721,-91.936,171.746,35.093,156.581
C04435=1053.108,201.472,-91.912,171.744,35.091,156.581
C04436=1053.103,201.223,-91.887,171.741,35.088,156.580
C04437=1053.096,200.975,-91.863,171.738,35.085,156.580
C04438=1053.090,200.726,-91.838,171.736,35.082,156.579
C04439=1053.084,200.478,-91.813,171.734,35.080,156.579
C04440=1053.078,200.229,-91.789,171.732,35.077,156.578
C04441=1053.072,199.979,-91.764,171.728,35.074,156.578
C04442=1053.065,199.731,-91.740,171.726,35.072,156.577
C04443=1053.060,199.483,-91.715,171.724,35.069,156.577
C04444=1053.054,199.233,-91.691,171.722,35.066,156.576
C04445=1053.047,198.986,-91.666,171.719,35.064,156.576
C04446=1053.041,198.736,-91.642,171.717,35.061,156.575
C04447=1053.035,198.487,-91.618,171.714,35.058,156.575
C04448=1053.030,198.239,-91.593,171.712,35.056,156.574
C04449=1053.023,197.990,-91.569,171.709,35.053,156.574
C04450=1053.017,197.741,-91.544,171.707,35.050,156.573
C04451=1053.011,197.493,-91.520,171.705,35.048,156.573
C04452=1053.005,197.244,-91.496,171.702,35.045,156.572
C04453=1052.999,196.996,-91.471,171.699,35.042,156.572
C04454=1052.993,196.747,-91.447,171.697,35.040,156.571
C04455=1052.987,196.497,-91.422,171.695,35.037,156.571
C04456=1052.981,196.249,-91.399,171.693,35.035,156.570
C04457=1052.975,196.000,-91.374,171.691,35.032,156.570
C04458=1052.968,195.752,-91.350,171.687,35.029,156.569
C04459=1052.962,195.503,-91.325,171.685,35.027,156.569
C04460=1052.957,195.253,-91.300,171.683,35.024,156.568
C04461=1052.951,195.005,-91.277,171.681,35.021,156.568
C04462=1052.945,194.756,-91.252,171.679,35.019,156.567
C04463=1052.939,194.508,-91.228,171.676,35.016,156.567
C04464=1052.933,194.258,-91.204,171.673,35.014,156.567
C04465=1052.927,194.010,-91.180,171.671,35.011,156.566
C04466=1052.920,193.761,-91.155,171.669,35.008,156.565
C04467=1052.914,193.513,-91.131,171.667,35.006,156.565
C04468=1052.909,193.264,-91.106,171.665,35.003,156.565
C04469=1052.902,193.016,-91.083,171.661,35.000,156.564
C04470=1052.897,192.766,-91.058,171.659,34.998,156.563
C04471=1052.891,192.518,-91.034,171.657,34.995,156.563
C04472=1052.885,192.269,-91.010,171.655,34.993,156.563
C04473=1052.879,192.020,-90.986,171.653,34.990,156.562
C04474=1052.873,191.771,-90.962,171.651,34.987,156.562
C04475=1052.867,191.523,-90.938,171.647,34.985,156.561
C04476=1052.861,191.274,-90.913,171.645,34.982,156.561
C04477=1052.855,191.025,-90.890,171.643,34.980,156.560
C04478=1052.849,190.777,-90.865,171.641,34.976,156.560
C04479=1052.842,190.492,-90.838,171.639,34.974,156.559
C04480=1052.836,190.208,-90.810,171.636,34.971,156.558
C04481=1052.829,189.924,-90.783,171.633,34.968,156.558
C04482=1052.822,189.639,-90.756,171.630,34.965,156.557
C04483=1052.817,189.391,-90.732,171.628,34.962,156.557
C04484=1052.810,189.142,-90.708,171.626,34.960,156.556
C04485=1052.805,188.893,-90.683,171.624,34.957,156.556
C04486=1052.798,188.644,-90.659,171.621,34.954,156.555
C04487=1052.793,188.396,-90.635,171.619,34.952,156.555
C04488=1052.787,188.147,-90.611,171.617,34.949,156.554
C04489=1052.781,187.897,-90.588,171.614,34.947,156.554
C04490=1052.775,187.649,-90.564,171.612,34.944,156.554
C04491=1052.769,187.401,-90.540,171.610,34.941,156.553
C04492=1052.763,187.152,-90.516,171.608,34.939,156.552
C04493=1052.757,186.903,-90.492,171.605,34.936,156.552
C04494=1052.752,186.654,-90.468,171.603,34.934,156.552
C04495=1052.746,186.405,-90.444,171.601,34.931,156.551
C04496=1052.740,186.157,-90.420,171.599,34.928,156.550
C04497=1052.734,185.908,-90.396,171.597,34.926,156.550
C04498=1052.729,185.658,-90.373,171.595,34.923,156.550
C04499=1052.723,185.410,-90.349,171.591,34.921,156.549
C04500=1052.717,185.162,-90.325,171.589,34.918,156.549
C04501=1052.711,184.913,-90.301,171.587,34.916,156.548
C04502=1052.705,184.664,-90.278,171.585,34.912,156.548
C04503=1052.700,184.415,-90.253,171.583,34.910,156.547
C04504=1052.693,184.166,-90.229,171.581,34.907,156.547
C04505=1052.687,183.917,-90.206,171.578,34.905,156.546
C04506=1052.681,183.669,-90.183,171.576,34.902,156.546
C04507=1052.675,183.419,-90.159,171.574,34.900,156.545
C04508=1052.669,183.171,-90.136,171.572,34.897,156.545
C04509=1052.663,182.921,-90.113,171.569,34.896,156.544
C04510=1052.657,182.673,-90.089,171.567,34.893,156.544
C04511=1052.651,182.425,-90.065,171.565,34.891,156.544
C04512=1052.644,182.175,-90.042,171.562,34.888,156.543
C04513=1052.638,181.927,-90.018,171.560,34.886,156.543
C04514=1052.632,181.678,-89.995,171.558,34.883,156.542
C04515=1052.626,181.429,-89.972,171.556,34.881,156.542
C04516=1052.620,181.180,-89.948,171.554,34.878,156.541
C04517=1052.614,180.932,-89.926,171.552,34.876,156.541
C04518=1052.607,180.683,-89.902,171.549,34.874,156.540
C04519=1052.601,180.434,-89.879,171.547,34.871,156.540
C04520=1052.595,180.186,-89.855,171.544,34.869,156.540
C04521=1052.589,179.936,-89.832,171.542,34.866,156.539
C04522=1052.583,179.688,-89.808,171.540,34.864,156.539
C04523=1052.577,179.439,-89.785,171.538,34.861,156.538
C04524=1052.571,179.189,-89.762,171.536,34.859,156.538
C04525=1052.565,178.941,-89.738,171.533,34.857,156.537
C04526=1052.559,178.692,-89.715,171.531,34.854,156.537
C04527=1052.553,178.442,-89.692,171.529,34.852,156.536
C04528=1052.547,178.194,-89.668,171.527,34.849,156.536
C04529=1052.540,177.946,-89.646,171.525,34.847,156.536
C04530=1052.534,177.697,-89.622,171.523,34.844,156.535
C04531=1052.528,177.448,-89.599,171.521,34.842,156.535
C04532=1052.522,177.199,-89.576,171.518,34.840,156.534
C04533=1052.516,176.950,-89.553,171.516,34.837,156.534
C04534=1052.510,176.702,-89.530,171.514,34.835,156.533
C04535=1052.504,176.452,-89.506,171.512,34.832,156.533
C04536=1052.498,176.203,-89.483,171.510,34.830,156.532
C04537=1052.491,175.955,-89.460,171.508,34.827,156.532
C04538=1052.486,175.706,-89.437,171.505,34.825,156.532
C04539=1052.479,175.457,-89.414,171.502,34.823,156.531
C04540=1052.474,175.208,-89.391,171.500,34.820,156.531
C04541=1052.468,174.959,-89.367,171.498,34.818,156.530
C04542=1052.462,174.711,-89.344,171.496,34.815,156.530
C04543=1052.455,174.426,-89.319,171.494,34.813,156.529
C04544=1052.448,174.141,-89.291,171.492,34.810,156.529
C04545=1052.441,173.857,-89.266,171.489,34.807,156.528
C04546=1052.435,173.572,-89.239,171.486,34.805,156.528
C04547=1052.428,173.323,-89.215,171.484,34.802,156.527
C04548=1052.422,173.074,-89.193,171.482,34.800,156.527
C04549=1052.416,172.826,-89.170,171.480,34.797,156.526
C04550=1052.410,172.577,-89.147,171.478,34.795,156.526
C04551=1052.405,172.328,-89.124,171.476,34.792,156.526
C04552=1052.399,172.079,-89.101,171.474,34.790,156.525
C04553=1052.393,171.830,-89.078,171.471,34.788,156.525
C04554=1052.386,171.581,-89.056,171.469,34.785,156.524
C04555=1052.380,171.332,-89.033,171.467,34.783,156.524
C04556=1052.374,171.084,-89.009,171.465,34.780,156.523
C04557=1052.369,170.835,-88.986,171.463,34.778,156.523
C04558=1052.363,170.586,-88.963,171.461,34.775,156.522
C04559=1052.357,170.337,-88.940,171.459,34.773,156.522
C04560=1052.351,170.088,-88.918,171.457,34.771,156.522
C04561=1052.345,169.839,-88.895,171.454,34.768,156.521
C04562=1052.339,169.590,-88.872,171.452,34.766,156.521
C04563=1052.333,169.342,-88.849,171.450,34.763,156.520
C04564=1052.328,169.093,-88.826,171.448,34.761,156.520
C04565=1052.322,168.844,-88.803,171.446,34.759,156.519
C04566=1052.315,168.594,-88.780,171.444,34.757,156.519
C04567=1052.309,168.346,-88.757,171.442,34.754,156.519
C04568=1052.303,168.097,-88.735,171.440,34.752,156.518
C04569=1052.298,167.848,-88.712,171.438,34.749,156.518
C04570=1052.292,167.599,-88.689,171.436,34.747,156.517
C04571=1052.286,167.350,-88.667,171.434,34.745,156.517
C04572=1052.280,167.101,-88.644,171.432,34.742,156.516
C04573=1052.274,166.852,-88.621,171.430,34.740,156.516
C04574=1052.269,166.603,-88.598,171.428,34.737,156.515
C04575=1052.263,166.354,-88.575,171.425,34.735,156.515
C04576=1052.256,166.105,-88.553,171.423,34.733,156.515
C04577=1052.251,165.857,-88.530,171.421,34.730,156.514
C04578=1052.245,165.608,-88.507,171.419,34.728,156.514
C04579=1052.239,165.359,-88.484,171.417,34.725,156.513
C04580=1052.233,165.110,-88.462,171.415,34.723,156.513
C04581=1052.227,164.861,-88.439,171.413,34.720,156.512
C04582=1052.222,164.612,-88.417,171.411,34.718,156.512
C04583=1052.217,164.364,-88.394,171.408,34.716,156.512
C04584=1052.210,164.115,-88.372,171.407,34.713,156.511
C04585=1052.204,163.866,-88.349,171.405,34.711,156.511
C04586=1052.199,163.617,-88.326,171.403,34.708,156.510
C04587=1052.193,163.368,-88.303,171.401,34.706,156.510
C04588=1052.187,163.119,-88.281,171.399,34.704,156.509
C04589=1052.181,162.870,-88.258,171.397,34.701,156.509
C04590=1052.176,162.621,-88.236,171.395,34.699,156.509
C04591=1052.170,162.372,-88.213,171.392,34.696,156.508
C04592=1052.164,162.123,-88.190,171.390,34.694,156.508
C04593=1052.158,161.874,-88.168,171.388,34.691,156.507
C04594=1052.152,161.625,-88.145,171.387,34.689,156.507
C04595=1052.147,161.377,-88.123,171.385,34.687,156.506
C04596=1052.141,161.128,-88.100,171.383,34.684,156.506
C04597=1052.135,160.879,-88.078,171.381,34.682,156.505
C04598=1052.129,160.630,-88.055,171.378,34.679,156.505
C04599=1052.123,160.381,-88.033,171.376,34.677,156.505
C04600=1052.118,160.132,-88.011,171.374,34.675,156.504
C04601=1052.111,159.883,-87.988,171.372,34.673,156.504
C04602=1052.105,159.634,-87.967,171.370,34.670,156.503
C04603=1052.099,159.385,-87.944,171.368,34.668,156.503
C04604=1052.093,159.136,-87.922,171.366,34.666,156.503
C04605=1052.087,158.887,-87.899,171.365,34.664,156.502
C04606=1052.081,158.638,-87.877,171.363,34.661,156.502
C04607=1052.074,158.353,-87.852,171.359,34.659,156.501
C04608=1052.068,158.068,-87.827,171.357,34.656,156.501
C04609=1052.060,157.783,-87.801,171.355,34.653,156.500
C04610=1052.054,157.498,-87.776,171.353,34.651,156.500
C04611=1052.048,157.249,-87.753,171.351,34.648,156.499
C04612=1052.042,157.000,-87.731,171.349,34.647,156.499
C04613=1052.035,156.751,-87.709,171.347,34.644,156.499
C04614=1052.030,156.502,-87.687,171.345,34.641,156.498
C04615=1052.024,156.254,-87.665,171.343,34.640,156.498
C04616=1052.018,156.004,-87.643,171.341,34.637,156.497
C04617=1052.012,155.756,-87.620,171.339,34.635,156.497
C04618=1052.006,155.506,-87.599,171.337,34.633,156.497
C04619=1052.000,155.257,-87.577,171.335,34.630,156.496
C04620=1051.994,155.008,-87.554,171.333,34.628,156.496
C04621=1051.988,154.759,-87.532,171.331,34.626,156.495
C04622=1051.981,154.510,-87.510,171.329,34.623,156.495
C04623=1051.976,154.262,-87.489,171.327,34.621,156.495
C04624=1051.970,154.012,-87.467,171.325,34.619,156.494
C04625=1051.964,153.764,-87.444,171.323,34.617,156.494
C04626=1051.958,153.515,-87.423,171.321,34.614,156.493
C04627=1051.952,153.265,-87.401,171.319,34.612,156.493
C04628=1051.946,153.017,-87.378,171.317,34.610,156.493
C04629=1051.940,152.768,-87.357,171.315,34.608,156.492
C04630=1051.934,152.519,-87.335,171.313,34.605,156.492
C04631=1051.928,152.270,-87.313,171.312,34.603,156.491
C04632=1051.921,152.021,-87.291,171.309,34.601,156.491
C04633=1051.916,151.772,-87.269,171.307,34.599,156.490
C04634=1051.910,151.522,-87.247,171.305,34.597,156.490
C04635=1051.904,151.274,-87.225,171.303,34.594,156.490
C04636=1051.898,151.025,-87.204,171.301,34.592,156.489
C04637=1051.892,150.776,-87.182,171.299,34.590,156.489
C04638=1051.886,150.527,-87.160,171.298,34.587,156.488
C04639=1051.881,150.278,-87.138,171.296,34.585,156.488
C04640=1051.874,150.029,-87.116,171.294,34.583,156.488
C04641=1051.868,149.780,-87.094,171.291,34.581,156.487
C04642=1051.862,149.531,-87.073,171.289,34.578,156.487
C04643=1051.856,149.282,-87.051,171.287,34.576,156.487
C04644=1051.851,149.033,-87.029,171.286,34.574,156.486
C04645=1051.844,148.784,-87.007,171.284,34.572,156.486
C04646=1051.838,148.535,-86.985,171.282,34.569,156.485
C04647=1051.832,148.286,-86.964,171.280,34.568,156.485
C04648=1051.827,148.037,-86.942,171.278,34.565,156.484
C04649=1051.820,147.788,-86.921,171.276,34.562,156.484
C04650=1051.814,147.539,-86.899,171.274,34.561,156.484
C04651=1051.808,147.290,-86.878,171.272,34.558,156.483
C04652=1051.803,147.041,-86.856,171.270,34.556,156.483
C04653=1051.796,146.792,-86.835,171.268,34.554,156.483
C04654=1051.790,146.543,-86.813,171.266,34.552,156.482
C04655=1051.784,146.294,-86.791,171.264,34.550,156.482
C04656=1051.778,146.046,-86.769,171.263,34.547,156.481
C04657=1051.772,145.797,-86.748,171.261,34.545,156.481
C04658=1051.766,145.547,-86.726,171.259,34.543,156.481
C04659=1051.760,145.298,-86.704,171.257,34.541,156.480
C04660=1051.754,145.050,-86.683,171.254,34.538,156.480
C04661=1051.748,144.801,-86.662,171.252,34.536,156.479
C04662=1051.742,144.551,-86.640,171.251,34.534,156.479
C04663=1051.736,144.302,-86.618,171.249,34.532,156.479
C04664=1051.730,144.053,-86.598,171.247,34.530,156.478
C04665=1051.723,143.804,-86.577,171.245,34.528,156.478
C04666=1051.717,143.555,-86.555,171.243,34.526,156.478
C04667=1051.712,143.306,-86.534,171.242,34.523,156.477
C04668=1051.706,143.057,-86.512,171.240,34.521,156.477
C04669=1051.699,142.808,-86.491,171.238,34.519,156.476
C04670=1051.694,142.559,-86.469,171.235,34.517,156.476
C04671=1051.687,142.274,-86.444,171.233,34.514,156.475
C04672=1051.680,141.988,-86.420,171.231,34.512,156.475
C04673=1051.673,141.703,-86.395,171.229,34.509,156.475
C04674=1051.667,141.418,-86.371,171.227,34.507,156.474
C04675=1051.660,141.169,-86.350,171.225,34.504,156.474
C04676=1051.654,140.920,-86.329,171.223,34.502,156.473
C04677=1051.648,140.671,-86.307,171.222,34.500,156.473
C04678=1051.642,140.422,-86.285,171.220,34.498,156.473
C04679=1051.636,140.173,-86.264,171.217,34.495,156.472
C04680=1051.630,139.924,-86.243,171.215,34.493,156.472
C04681=1051.624,139.674,-86.222,171.213,34.491,156.471
C04682=1051.619,139.426,-86.200,171.212,34.489,156.471
C04683=1051.612,139.177,-86.179,171.210,34.487,156.471
C04684=1051.606,138.928,-86.158,171.208,34.484,156.470
C04685=1051.601,138.678,-86.137,171.206,34.483,156.470
C04686=1051.594,138.429,-86.116,171.204,34.480,156.469
C04687=1051.588,138.181,-86.095,171.203,34.478,156.469
C04688=1051.582,137.932,-86.073,171.201,34.476,156.469
C04689=1051.576,137.682,-86.052,171.198,34.474,156.468
C04690=1051.571,137.434,-86.031,171.196,34.472,156.468
C04691=1051.564,137.185,-86.010,171.195,34.469,156.467
C04692=1051.558,136.935,-85.989,171.193,34.467,156.467
C04693=1051.552,136.686,-85.968,171.191,34.465,156.467
C04694=1051.545,136.437,-85.947,171.189,34.463,156.466
C04695=1051.540,136.188,-85.926,171.187,34.461,156.466
C04696=1051.534,135.939,-85.905,171.186,34.458,156.466
C04697=1051.528,135.691,-85.883,171.184,34.457,156.465
C04698=1051.522,135.441,-85.863,171.182,34.455,156.465
C04699=1051.516,135.192,-85.841,171.180,34.452,156.464
C04700=1051.510,134.943,-85.820,171.178,34.450,156.464
C04701=1051.503,134.694,-85.800,171.176,34.448,156.464
C04702=1051.498,134.445,-85.778,171.174,34.446,156.463
C04703=1051.492,134.195,-85.758,171.172,34.444,156.463
C04704=1051.486,133.947,-85.737,171.171,34.441,156.463
C04705=1051.480,133.698,-85.715,171.169,34.439,156.462
C04706=1051.474,133.449,-85.695,171.167,34.437,156.462
C04707=1051.467,133.200,-85.674,171.165,34.435,156.461
C04708=1051.462,132.951,-85.653,171.164,34.433,156.461
C04709=1051.456,132.702,-85.631,171.162,34.430,156.461
C04710=1051.449,132.452,-85.611,171.159,34.428,156.460
C04711=1051.444,132.204,-85.590,171.157,34.426,156.460
C04712=1051.438,131.954,-85.569,171.156,34.424,156.460
C04713=1051.432,131.706,-85.548,171.154,34.422,156.459
C04714=1051.426,131.456,-85.527,171.152,34.420,156.459
C04715=1051.419,131.208,-85.507,171.150,34.418,156.458
C04716=1051.414,130.958,-85.486,171.149,34.416,156.458
C04717=1051.407,130.710,-85.465,171.147,34.413,156.458
C04718=1051.401,130.460,-85.445,171.145,34.411,156.457
C04719=1051.395,130.211,-85.424,171.143,34.409,156.457
C04720=1051.389,129.962,-85.403,171.142,34.407,156.457
C04721=1051.382,129.713,-85.383,171.139,34.405,156.456
C04722=1051.376,129.464,-85.362,171.137,34.403,156.456
C04723=1051.370,129.215,-85.341,171.135,34.401,156.456
C04724=1051.365,128.965,-85.321,171.134,34.399,156.455
C04725=1051.358,128.717,-85.300,171.132,34.397,156.455
C04726=1051.352,128.468,-85.280,171.130,34.395,156.454
C04727=1051.346,128.218,-85.259,171.128,34.393,156.454
C04728=1051.340,127.970,-85.238,171.127,34.391,156.454
C04729=1051.333,127.720,-85.218,171.125,34.388,156.453
C04730=1051.328,127.471,-85.197,171.123,34.386,156.453
C04731=1051.321,127.222,-85.176,171.121,34.384,156.453
C04732=1051.315,126.973,-85.156,171.120,34.383,156.452
C04733=1051.309,126.724,-85.135,171.117,34.380,156.452
C04734=1051.303,126.475,-85.115,171.115,34.378,156.452
C04735=1051.296,126.189,-85.092,171.113,34.376,156.451
C04736=1051.289,125.904,-85.068,171.111,34.373,156.451
C04737=1051.282,125.619,-85.044,171.109,34.371,156.450
C04738=1051.275,125.333,-85.021,171.107,34.369,156.450
C04739=1051.268,125.084,-85.000,171.105,34.367,156.450
C04740=1051.263,124.835,-84.980,171.104,34.364,156.449
C04741=1051.256,124.585,-84.960,171.102,34.362,156.449
C04742=1051.250,124.337,-84.939,171.100,34.360,156.448
C04743=1051.244,124.087,-84.918,171.099,34.358,156.448
C04744=1051.238,123.838,-84.898,171.096,34.356,156.448
C04745=1051.232,123.589,-84.878,171.094,34.354,156.447
C04746=1051.226,123.340,-84.857,171.092,34.352,156.447
C04747=1051.220,123.091,-84.836,171.091,34.349,156.447
C04748=1051.214,122.842,-84.816,171.089,34.347,156.446
C04749=1051.208,122.593,-84.796,171.087,34.345,156.446
C04750=1051.202,122.344,-84.776,171.086,34.343,156.445
C04751=1051.196,122.094,-84.755,171.084,34.341,156.445
C04752=1051.190,121.845,-84.735,171.082,34.339,156.445
C04753=1051.184,121.596,-84.714,171.080,34.337,156.444
C04754=1051.178,121.348,-84.694,171.079,34.335,156.444
C04755=1051.172,121.098,-84.673,171.077,34.333,156.444
C04756=1051.166,120.849,-84.653,171.074,34.331,156.443
C04757=1051.160,120.600,-84.633,171.073,34.328,156.443
C04758=1051.154,120.351,-84.613,171.071,34.326,156.443
C04759=1051.148,120.101,-84.592,171.069,34.324,156.442
C04760=1051.142,119.853,-84.572,171.068,34.322,156.442
C04761=1051.136,119.604,-84.552,171.066,34.320,156.441
C04762=1051.130,119.354,-84.531,171.064,34.318,156.441
C04763=1051.124,119.105,-84.511,171.062,34.315,156.441
C04764=1051.118,118.856,-84.491,171.061,34.314,156.440
C04765=1051.111,118.607,-84.471,171.059,34.312,156.440
C04766=1051.106,118.358,-84.450,171.057,34.309,156.440
C04767=1051.100,118.109,-84.430,171.056,34.307,156.439
C04768=1051.094,117.859,-84.410,171.053,34.305,156.439
C04769=1051.088,117.610,-84.389,171.051,34.303,156.438
C04770=1051.082,117.362,-84.370,171.050,34.301,156.438
C04771=1051.076,117.113,-84.350,171.048,34.299,156.438
C04772=1051.070,116.863,-84.329,171.046,34.296,156.437
C04773=1051.065,116.614,-84.309,171.045,34.294,156.437
C04774=1051.059,116.365,-84.289,171.043,34.292,156.437
C04775=1051.052,116.116,-84.268,171.041,34.290,156.436
C04776=1051.046,115.867,-84.248,171.040,34.288,156.436
C04777=1051.041,115.618,-84.228,171.038,34.286,156.436
C04778=1051.035,115.369,-84.208,171.036,34.284,156.435
C04779=1051.028,115.119,-84.188,171.035,34.282,156.435
C04780=1051.022,114.871,-84.168,171.033,34.280,156.434
C04781=1051.017,114.622,-84.147,171.030,34.277,156.434
C04782=1051.011,114.373,-84.127,171.029,34.275,156.434
C04783=1051.005,114.124,-84.107,171.027,34.273,156.433
C04784=1050.999,113.874,-84.088,171.025,34.271,156.433
C04785=1050.993,113.625,-84.068,171.024,34.269,156.433
C04786=1050.987,113.376,-84.047,171.022,34.267,156.432
C04787=1050.981,113.126,-84.027,171.020,34.265,156.432
C04788=1050.975,112.878,-84.007,171.019,34.262,156.431
C04789=1050.969,112.628,-83.988,171.017,34.260,156.431
C04790=1050.963,112.379,-83.968,171.015,34.259,156.431
C04791=1050.956,112.130,-83.947,171.014,34.257,156.430
C04792=1050.950,111.881,-83.927,171.012,34.254,156.430
C04793=1050.944,111.632,-83.907,171.010,34.252,156.430
C04794=1050.939,111.383,-83.888,171.008,34.250,156.429
C04795=1050.932,111.133,-83.868,171.006,34.248,156.429
C04796=1050.926,110.884,-83.848,171.004,34.246,156.429
C04797=1050.919,110.636,-83.828,171.003,34.244,156.428
C04798=1050.914,110.386,-83.809,171.001,34.242,156.428
C04799=1050.907,110.100,-83.786,170.999,34.239,156.427
C04800=1050.899,109.815,-83.763,170.997,34.237,156.427
C04801=1050.893,109.529,-83.740,170.995,34.235,156.427
C04802=1050.885,109.244,-83.718,170.993,34.233,156.426
C04803=1050.879,108.994,-83.699,170.991,34.230,156.426
C04804=1050.873,108.745,-83.679,170.990,34.228,156.426
C04805=1050.867,108.497,-83.659,170.988,34.226,156.425
C04806=1050.861,108.246,-83.639,170.986,34.224,156.425
C04807=1050.854,107.998,-83.620,170.984,34.223,156.425
C04808=1050.848,107.749,-83.600,170.982,34.221,156.424
C04809=1050.843,107.500,-83.581,170.980,34.218,156.424
C04810=1050.837,107.251,-83.561,170.979,34.216,156.423
C04811=1050.831,107.001,-83.541,170.977,34.214,156.423
C04812=1050.825,106.752,-83.521,170.975,34.212,156.423
C04813=1050.818,106.503,-83.502,170.974,34.210,156.422
C04814=1050.812,106.254,-83.482,170.972,34.208,156.422
C04815=1050.806,106.005,-83.462,170.970,34.206,156.422
C04816=1050.800,105.755,-83.443,170.969,34.204,156.421
C04817=1050.794,105.506,-83.423,170.967,34.202,156.421
C04818=1050.788,105.257,-83.404,170.966,34.200,156.421
C04819=1050.781,105.008,-83.384,170.964,34.198,156.420
C04820=1050.776,104.759,-83.365,170.962,34.196,156.420
C04821=1050.770,104.510,-83.345,170.960,34.194,156.420
C04822=1050.764,104.261,-83.326,170.958,34.192,156.419
C04823=1050.757,104.011,-83.306,170.956,34.190,156.419
C04824=1050.752,103.762,-83.286,170.955,34.187,156.419
C04825=1050.745,103.513,-83.267,170.953,34.185,156.418
C04826=1050.739,103.264,-83.248,170.951,34.183,156.418
C04827=1050.733,103.015,-83.228,170.950,34.181,156.418
C04828=1050.728,102.765,-83.208,170.948,34.179,156.417
C04829=1050.722,102.517,-83.189,170.946,34.177,156.417
C04830=1050.715,102.268,-83.170,170.945,34.175,156.416
C04831=1050.709,102.019,-83.150,170.943,34.173,156.416
C04832=1050.703,101.769,-83.130,170.941,34.171,156.416
C04833=1050.697,101.519,-83.111,170.940,34.169,156.415
C04834=1050.691,101.270,-83.091,170.938,34.167,156.415
C04835=1050.685,101.021,-83.072,170.936,34.165,156.415
C04836=1050.679,100.772,-83.052,170.934,34.163,156.414
C04837=1050.673,100.523,-83.033,170.932,34.161,156.414
C04838=1050.667,100.274,-83.015,170.931,34.158,156.414
C04839=1050.661,100.025,-82.995,170.929,34.156,156.413
C04840=1050.655,99.776,-82.975,170.927,34.154,156.413
C04841=1050.648,99.526,-82.956,170.926,34.153,156.413
C04842=1050.642,99.277,-82.936,170.924,34.151,156.412
C04843=1050.636,99.028,-82.918,170.922,34.149,156.412
C04844=1050.630,98.778,-82.899,170.921,34.147,156.412
C04845=1050.623,98.530,-82.879,170.919,34.145,156.411
C04846=1050.617,98.280,-82.860,170.917,34.143,156.411
C04847=1050.611,98.031,-82.841,170.916,34.140,156.410
C04848=1050.605,97.782,-82.822,170.914,34.138,156.410
C04849=1050.599,97.533,-82.802,170.912,34.136,156.410
C04850=1050.593,97.284,-82.783,170.911,34.134,156.410
C04851=1050.587,97.035,-82.764,170.908,34.132,156.409
C04852=1050.581,96.785,-82.746,170.907,34.131,156.409
C04853=1050.574,96.536,-82.725,170.905,34.129,156.409
C04854=1050.568,96.287,-82.707,170.903,34.127,156.408
C04855=1050.562,96.037,-82.687,170.902,34.124,156.408
C04856=1050.556,95.788,-82.669,170.900,34.122,156.407
C04857=1050.550,95.539,-82.649,170.898,34.120,156.407
C04858=1050.543,95.290,-82.630,170.897,34.118,156.407
C04859=1050.538,95.041,-82.611,170.895,34.116,156.406
C04860=1050.532,94.791,-82.592,170.893,34.114,156.406
C04861=1050.525,94.542,-82.573,170.892,34.113,156.406
C04862=1050.520,94.293,-82.554,170.890,34.110,156.405
C04863=1050.513,94.008,-82.532,170.888,34.108,156.405
C04864=1050.506,93.722,-82.510,170.886,34.105,156.405
C04865=1050.499,93.437,-82.488,170.885,34.103,156.404
C04866=1050.492,93.150,-82.466,170.882,34.101,156.404
C04867=1050.485,92.902,-82.447,170.880,34.099,156.404
C04868=1050.479,92.652,-82.428,170.878,34.097,156.403
C04869=1050.473,92.403,-82.409,170.877,34.095,156.403
C04870=1050.467,92.154,-82.390,170.875,34.093,156.402
C04871=1050.461,91.905,-82.371,170.874,34.091,156.402
C04872=1050.455,91.655,-82.352,170.872,34.089,156.402
C04873=1050.449,91.406,-82.333,170.870,34.087,156.401
C04874=1050.443,91.157,-82.314,170.869,34.085,156.401
C04875=1050.437,90.908,-82.296,170.867,34.083,156.401
C04876=1050.432,90.659,-82.277,170.865,34.080,156.400
C04877=1050.425,90.410,-82.258,170.864,34.078,156.400
C04878=1050.419,90.160,-82.239,170.862,34.076,156.400
C04879=1050.413,89.911,-82.220,170.861,34.074,156.399
C04880=1050.407,89.662,-82.201,170.859,34.072,156.399
C04881=1050.400,89.413,-82.183,170.857,34.071,156.399
C04882=1050.394,89.163,-82.164,170.855,34.069,156.398
C04883=1050.388,88.914,-82.145,170.853,34.067,156.398
C04884=1050.382,88.665,-82.126,170.851,34.065,156.398
C04885=1050.375,88.416,-82.108,170.850,34.063,156.397
C04886=1050.370,88.167,-82.088,170.848,34.061,156.397
C04887=1050.363,87.918,-82.070,170.846,34.059,156.397
C04888=1050.357,87.668,-82.051,170.845,34.057,156.396
C04889=1050.350,87.419,-82.032,170.843,34.055,156.396
C04890=1050.345,87.170,-82.013,170.842,34.053,156.396
C04891=1050.338,86.920,-81.995,170.840,34.051,156.395
C04892=1050.332,86.671,-81.977,170.838,34.049,156.395
C04893=1050.326,86.422,-81.958,170.837,34.047,156.395
C04894=1050.320,86.172,-81.939,170.835,34.045,156.394
C04895=1050.313,85.923,-81.920,170.833,34.043,156.394
C04896=1050.307,85.674,-81.901,170.832,34.041,156.394
C04897=1050.301,85.425,-81.883,170.830,34.039,156.393
C04898=1050.295,85.175,-81.865,170.829,34.037,156.393
C04899=1050.289,84.927,-81.846,170.827,34.035,156.393
C04900=1050.283,84.677,-81.827,170.824,34.033,156.392
C04901=1050.277,84.428,-81.809,170.823,34.031,156.392
C04902=1050.270,84.179,-81.790,170.821,34.029,156.392
C04903=1050.264,83.930,-81.771,170.819,34.027,156.391
C04904=1050.258,83.680,-81.753,170.818,34.025,156.391
C04905=1050.252,83.431,-81.734,170.816,34.023,156.391
C04906=1050.245,83.182,-81.716,170.815,34.021,156.390
C04907=1050.240,82.933,-81.697,170.813,34.019,156.390
C04908=1050.234,82.683,-81.679,170.811,34.017,156.390
C04909=1050.228,82.434,-81.660,170.810,34.015,156.389
C04910=1050.221,82.185,-81.641,170.808,34.013,156.389
C04911=1050.215,81.936,-81.623,170.806,34.011,156.389
C04912=1050.209,81.686,-81.605,170.805,34.009,156.388
C04913=1050.203,81.437,-81.586,170.803,34.007,156.388
C04914=1050.197,81.188,-81.567,170.802,34.005,156.388
C04915=1050.191,80.939,-81.549,170.800,34.003,156.387
C04916=1050.185,80.690,-81.531,170.798,34.001,156.387
C04917=1050.178,80.440,-81.512,170.797,33.999,156.387
C04918=1050.173,80.191,-81.493,170.795,33.997,156.386
C04919=1050.167,79.942,-81.475,170.793,33.995,156.386
C04920=1050.161,79.693,-81.457,170.791,33.993,156.386
C04921=1050.154,79.444,-81.438,170.789,33.991,156.385
C04922=1050.148,79.194,-81.420,170.788,33.989,156.385
C04923=1050.142,78.945,-81.401,170.786,33.987,156.385
C04924=1050.137,78.696,-81.383,170.785,33.985,156.384
C04925=1050.131,78.446,-81.365,170.783,33.983,156.384
C04926=1050.124,78.197,-81.346,170.781,33.981,156.384
C04927=1050.117,77.912,-81.325,170.779,33.978,156.383
C04928=1050.110,77.626,-81.304,170.778,33.977,156.383
C04929=1050.103,77.340,-81.284,170.776,33.974,156.383
C04930=1050.096,77.054,-81.262,170.774,33.972,156.382
C04931=1050.090,76.805,-81.244,170.772,33.970,156.382
C04932=1050.084,76.555,-81.226,170.771,33.968,156.382
C04933=1050.077,76.306,-81.207,170.769,33.966,156.381
C04934=1050.071,76.057,-81.190,170.767,33.964,156.381
C04935=1050.065,75.808,-81.172,170.766,33.962,156.381
C04936=1050.058,75.559,-81.153,170.764,33.960,156.380
C04937=1050.052,75.309,-81.135,170.762,33.958,156.380
C04938=1050.046,75.060,-81.116,170.760,33.956,156.380
C04939=1050.040,74.811,-81.099,170.758,33.954,156.379
C04940=1050.034,74.561,-81.081,170.757,33.952,156.379
C04941=1050.028,74.312,-81.062,170.755,33.951,156.379
C04942=1050.021,74.063,-81.044,170.753,33.949,156.378
C04943=1050.016,73.814,-81.026,170.752,33.947,156.378
C04944=1050.009,73.564,-81.008,170.750,33.945,156.378
C04945=1050.003,73.315,-80.989,170.749,33.943,156.377
C04946=1049.997,73.066,-80.971,170.747,33.941,156.377
C04947=1049.991,72.817,-80.953,170.745,33.938,156.377
C04948=1049.985,72.567,-80.935,170.744,33.936,156.376
C04949=1049.978,72.318,-80.918,170.742,33.934,156.376
C04950=1049.972,72.069,-80.899,170.740,33.932,156.376
C04951=1049.966,71.820,-80.882,170.739,33.930,156.375
C04952=1049.960,71.571,-80.863,170.737,33.928,156.375
C04953=1049.954,71.321,-80.845,170.736,33.926,156.375
C04954=1049.948,71.072,-80.828,170.734,33.925,156.374
C04955=1049.942,70.823,-80.809,170.732,33.923,156.374
C04956=1049.936,70.573,-80.791,170.731,33.921,156.374
C04957=1049.929,70.324,-80.774,170.729,33.919,156.373
C04958=1049.923,70.075,-80.755,170.727,33.917,156.373
C04959=1049.917,69.825,-80.737,170.725,33.915,156.373
C04960=1049.911,69.576,-80.720,170.723,33.913,156.372
C04961=1049.905,69.327,-80.701,170.722,33.911,156.372
C04962=1049.899,69.078,-80.683,170.720,33.909,156.372
C04963=1049.892,68.828,-80.666,170.718,33.907,156.371
C04964=1049.886,68.580,-80.648,170.717,33.905,156.371
C04965=1049.880,68.330,-80.630,170.715,33.903,156.371
C04966=1049.874,68.080,-80.612,170.714,33.901,156.370
C04967=1049.867,67.831,-80.594,170.712,33.899,156.370
C04968=1049.861,67.582,-80.576,170.710,33.897,156.370
C04969=1049.855,67.333,-80.558,170.709,33.895,156.369
C04970=1049.849,67.083,-80.540,170.707,33.893,156.369
C04971=1049.843,66.834,-80.523,170.705,33.891,156.369
C04972=1049.836,66.584,-80.505,170.704,33.890,156.369
C04973=1049.830,66.335,-80.487,170.702,33.888,156.368
C04974=1049.824,66.087,-80.470,170.701,33.886,156.368
C04975=1049.818,65.837,-80.452,170.699,33.884,156.368
C04976=1049.812,65.587,-80.434,170.697,33.882,156.367
C04977=1049.806,65.338,-80.416,170.696,33.880,156.367
C04978=1049.799,65.089,-80.398,170.694,33.878,156.367
C04979=1049.793,64.840,-80.381,170.692,33.876,156.366
C04980=1049.787,64.590,-80.363,170.691,33.874,156.366
C04981=1049.780,64.341,-80.345,170.689,33.872,156.366
C04982=1049.775,64.092,-80.328,170.687,33.870,156.365
C04983=1049.768,63.843,-80.311,170.685,33.868,156.365
C04984=1049.762,63.593,-80.293,170.683,33.866,156.365
C04985=1049.756,63.344,-80.276,170.682,33.864,156.364
C04986=1049.750,63.094,-80.258,170.680,33.863,156.364
C04987=1049.743,62.845,-80.240,170.678,33.861,156.364
C04988=1049.737,62.596,-80.222,170.677,33.859,156.364
C04989=1049.730,62.347,-80.205,170.675,33.857,156.363
C04990=1049.724,62.097,-80.187,170.673,33.855,156.363
C04991=1049.718,61.883,-80.172,170.672,33.854,156.363
C04992=1049.713,61.669,-80.158,170.671,33.852,156.362
C04993=1049.707,61.454,-80.143,170.669,33.851,156.362
C04994=1049.702,61.240,-80.128,170.668,33.849,156.362
C04995=1049.697,61.026,-80.112,170.666,33.847,156.362
C04996=1049.691,60.811,-80.097,170.665,33.845,156.361
C04997=1049.686,60.597,-80.082,170.664,33.844,156.361
C04998=1049.680,60.383,-80.068,170.662,33.843,156.361
C04999=1049.674,60.133,-80.050,170.660,33.841,156.361
C05000=1049.668,59.885,-80.033,170.659,33.839,156.360
C05001=1049.662,59.635,-80.015,170.657,33.837,156.360
C05002=1049.655,59.385,-79.997,170.656,33.835,156.360
C05003=1049.649,59.137,-79.980,170.654,33.833,156.359
C05004=1049.643,58.887,-79.963,170.652,33.831,156.359
C05005=1049.636,58.638,-79.946,170.651,33.830,156.359
C05006=1049.630,58.388,-79.928,170.649,33.828,156.358
C05007=1049.624,58.138,-79.911,170.647,33.826,156.358
C05008=1049.617,57.890,-79.894,170.646,33.824,156.358
C05009=1049.611,57.640,-79.876,170.644,33.822,156.357
C05010=1049.605,57.391,-79.859,170.641,33.820,156.357
C05011=1049.599,57.141,-79.841,170.640,33.818,156.357
C05012=1049.593,56.893,-79.824,170.638,33.816,156.357
C05013=1049.586,56.643,-79.806,170.637,33.815,156.356
C05014=1049.580,56.394,-79.789,170.635,33.813,156.356
C05015=1049.573,56.145,-79.772,170.633,33.811,156.356
C05016=1049.568,55.894,-79.755,170.632,33.809,156.355
C05017=1049.561,55.646,-79.738,170.630,33.807,156.355
C05018=1049.554,55.396,-79.720,170.628,33.805,156.355
C05019=1049.549,55.147,-79.703,170.627,33.803,156.354
C05020=1049.542,54.898,-79.686,170.625,33.801,156.354
C05021=1049.537,54.649,-79.668,170.623,33.799,156.354
C05022=1049.530,54.399,-79.651,170.622,33.797,156.354
C05023=1049.524,54.150,-79.634,170.620,33.795,156.353
C05024=1049.518,53.900,-79.616,170.619,33.794,156.353
C05025=1049.511,53.652,-79.599,170.617,33.792,156.353
C05026=1049.506,53.401,-79.582,170.615,33.790,156.352
C05027=1049.499,53.152,-79.565,170.614,33.788,156.352
C05028=1049.492,52.903,-79.548,170.612,33.786,156.352
C05029=1049.487,52.654,-79.530,170.610,33.784,156.351
C05030=1049.480,52.404,-79.514,170.609,33.782,156.351
C05031=1049.474,52.155,-79.497,170.607,33.780,156.351
C05032=1049.469,51.906,-79.479,170.605,33.778,156.350
C05033=1049.462,51.657,-79.462,170.604,33.776,156.350
C05034=1049.456,51.407,-79.446,170.602,33.774,156.350
C05035=1049.450,51.158,-79.428,170.601,33.772,156.350
C05036=1049.443,50.909,-79.411,170.599,33.770,156.349
C05037=1049.437,50.659,-79.394,170.597,33.768,156.349
C05038=1049.431,50.410,-79.377,170.595,33.767,156.349
C05039=1049.424,50.160,-79.359,170.593,33.765,156.348
C05040=1049.419,49.911,-79.342,170.591,33.763,156.348
C05041=1049.413,49.662,-79.325,170.590,33.761,156.348
C05042=1049.406,49.413,-79.308,170.588,33.759,156.347
C05043=1049.401,49.163,-79.291,170.586,33.757,156.347
C05044=1049.394,48.913,-79.274,170.585,33.755,156.347
C05045=1049.388,48.665,-79.257,170.583,33.753,156.346
C05046=1049.383,48.415,-79.240,170.582,33.751,156.346
C05047=1049.373,48.059,-79.216,170.579,33.749,156.346
C05048=1049.364,47.704,-79.191,170.577,33.746,156.345
C05049=1049.356,47.347,-79.166,170.575,33.743,156.345
C05050=1049.347,46.991,-79.143,170.572,33.740,156.344
C05051=1049.341,46.743,-79.126,170.571,33.738,156.344
C05052=1049.335,46.493,-79.108,170.569,33.736,156.344
C05053=1049.329,46.244,-79.092,170.567,33.735,156.343
C05054=1049.322,45.994,-79.075,170.566,33.733,156.343
C05055=1049.315,45.708,-79.055,170.564,33.730,156.343
C05056=1049.308,45.422,-79.035,170.562,33.728,156.342
C05057=1049.302,45.135,-79.016,170.560,33.726,156.342
C05058=1049.294,44.850,-78.997,170.558,33.724,156.342
C05059=1049.289,44.600,-78.980,170.557,33.722,156.341
C05060=1049.283,44.351,-78.963,170.555,33.720,156.341
C05061=1049.276,44.101,-78.946,170.553,33.718,156.341
C05062=1049.270,43.852,-78.929,170.552,33.716,156.340
C05063=1049.265,43.603,-78.912,170.550,33.714,156.340
C05064=1049.259,43.353,-78.896,170.548,33.712,156.340
C05065=1049.252,43.104,-78.879,170.547,33.711,156.340
C05066=1049.246,42.855,-78.863,170.545,33.709,156.339
C05067=1049.239,42.605,-78.845,170.543,33.707,156.339
C05068=1049.233,42.356,-78.829,170.541,33.705,156.339
C05069=1049.227,42.107,-78.812,170.539,33.703,156.338
C05070=1049.220,41.857,-78.795,170.537,33.701,156.338
C05071=1049.215,41.607,-78.779,170.536,33.699,156.338
C05072=1049.209,41.359,-78.762,170.534,33.697,156.337
C05073=1049.202,41.109,-78.745,170.532,33.695,156.337
C05074=1049.196,40.859,-78.729,170.531,33.693,156.337
C05075=1049.190,40.611,-78.712,170.529,33.692,156.337
C05076=1049.184,40.361,-78.696,170.527,33.690,156.336
C05077=1049.177,40.111,-78.679,170.526,33.688,156.336
C05078=1049.171,39.862,-78.662,170.524,33.686,156.336
C05079=1049.165,39.613,-78.646,170.522,33.684,156.335
C05080=1049.159,39.363,-78.629,170.521,33.682,156.335
C05081=1049.152,39.114,-78.612,170.519,33.681,156.335
C05082=1049.146,38.865,-78.596,170.517,33.679,156.335
C05083=1049.141,38.616,-78.580,170.516,33.677,156.334
C05084=1049.134,38.366,-78.562,170.514,33.675,156.334
C05085=1049.128,38.117,-78.546,170.513,33.673,156.334
C05086=1049.122,37.867,-78.530,170.511,33.671,156.333
C05087=1049.116,37.618,-78.513,170.509,33.669,156.333
C05088=1049.109,37.369,-78.496,170.508,33.668,156.333
C05089=1049.103,37.119,-78.480,170.506,33.666,156.332
C05090=1049.097,36.870,-78.464,170.504,33.664,156.332
C05091=1049.090,36.620,-78.447,170.502,33.662,156.332
C05092=1049.085,36.371,-78.431,170.501,33.660,156.332
C05093=1049.078,36.122,-78.414,170.499,33.658,156.331
C05094=1049.071,35.872,-78.398,170.497,33.657,156.331
C05095=1049.065,35.623,-78.381,170.496,33.655,156.331
C05096=1049.059,35.373,-78.365,170.494,33.653,156.330
C05097=1049.053,35.124,-78.349,170.492,33.651,156.330
C05098=1049.047,34.874,-78.332,170.491,33.650,156.330
C05099=1049.040,34.626,-78.316,170.489,33.648,156.330
C05100=1049.034,34.376,-78.300,170.487,33.646,156.329
C05101=1049.028,34.127,-78.283,170.486,33.644,156.329
C05102=1049.021,33.877,-78.267,170.484,33.642,156.329
C05103=1049.015,33.628,-78.251,170.482,33.640,156.328
C05104=1049.009,33.378,-78.234,170.481,33.638,156.328
C05105=1049.003,33.129,-78.219,170.479,33.637,156.328
C05106=1048.997,32.880,-78.202,170.477,33.635,156.328
C05107=1048.990,32.630,-78.186,170.476,33.633,156.327
C05108=1048.984,32.380,-78.169,170.474,33.632,156.327
C05109=1048.978,32.132,-78.153,170.472,33.630,156.327
C05110=1048.971,31.883,-78.137,170.471,33.628,156.326
C05111=1048.965,31.633,-78.121,170.468,33.626,156.326
C05112=1048.959,31.383,-78.104,170.466,33.624,156.326
C05113=1048.953,31.134,-78.088,170.465,33.622,156.326
C05114=1048.947,30.885,-78.071,170.463,33.620,156.325
C05115=1048.941,30.635,-78.055,170.461,33.618,156.325
C05116=1048.934,30.386,-78.040,170.459,33.617,156.325
C05117=1048.928,30.137,-78.023,170.458,33.615,156.324
C05118=1048.922,29.887,-78.007,170.456,33.613,156.324
C05119=1048.915,29.601,-77.988,170.454,33.611,156.324
C05120=1048.907,29.315,-77.970,170.452,33.609,156.324
C05121=1048.900,29.028,-77.952,170.450,33.607,156.323
C05122=1048.894,28.742,-77.933,170.448,33.605,156.323
C05123=1048.887,28.492,-77.917,170.447,33.603,156.323
C05124=1048.881,28.243,-77.901,170.445,33.601,156.322
C05125=1048.875,27.994,-77.884,170.443,33.600,156.322
C05126=1048.868,27.745,-77.869,170.442,33.598,156.322
C05127=1048.862,27.495,-77.852,170.440,33.596,156.321
C05128=1048.856,27.245,-77.836,170.438,33.594,156.321
C05129=1048.849,26.996,-77.820,170.436,33.592,156.321
C05130=1048.844,26.746,-77.805,170.435,33.590,156.321
C05131=1048.837,26.497,-77.789,170.433,33.589,156.320
C05132=1048.831,26.248,-77.773,170.431,33.587,156.320
C05133=1048.825,25.999,-77.757,170.430,33.585,156.320
C05134=1048.818,25.749,-77.740,170.428,33.584,156.320
C05135=1048.812,25.500,-77.724,170.426,33.581,156.319
C05136=1048.805,25.250,-77.709,170.425,33.580,156.319
C05137=1048.799,25.001,-77.693,170.423,33.578,156.319
C05138=1048.793,24.751,-77.677,170.421,33.576,156.318
C05139=1048.787,24.502,-77.661,170.419,33.574,156.318
C05140=1048.781,24.253,-77.645,170.418,33.573,156.318
C05141=1048.774,24.004,-77.629,170.416,33.571,156.318
C05142=1048.768,23.754,-77.614,170.414,33.569,156.317
C05143=1048.761,23.504,-77.598,170.413,33.567,156.317
C05144=1048.755,23.255,-77.581,170.411,33.565,156.317
C05145=1048.749,23.006,-77.566,170.409,33.564,156.317
C05146=1048.743,22.756,-77.550,170.407,33.562,156.316
C05147=1048.737,22.506,-77.534,170.406,33.560,156.316
C05148=1048.730,22.257,-77.518,170.404,33.559,156.316
C05149=1048.724,22.008,-77.502,170.402,33.557,156.315
C05150=1048.718,21.758,-77.487,170.401,33.555,156.315
C05151=1048.712,21.509,-77.471,170.399,33.553,156.315
C05152=1048.705,21.260,-77.455,170.397,33.551,156.315
C05153=1048.700,21.010,-77.440,170.395,33.550,156.314
C05154=1048.693,20.761,-77.424,170.394,33.548,156.314
C05155=1048.687,20.512,-77.408,170.392,33.546,156.314
C05156=1048.681,20.262,-77.391,170.390,33.545,156.314
C05157=1048.675,20.013,-77.376,170.389,33.543,156.313
C05158=1048.668,19.764,-77.361,170.387,33.541,156.313
C05159=1048.662,19.514,-77.345,170.385,33.539,156.313
C05160=1048.655,19.264,-77.329,170.383,33.537,156.312
C05161=1048.649,19.014,-77.313,170.382,33.536,156.312
C05162=1048.643,18.765,-77.298,170.380,33.534,156.312
C05163=1048.637,18.515,-77.282,170.378,33.532,156.312
C05164=1048.630,18.266,-77.267,170.376,33.530,156.311
C05165=1048.624,18.017,-77.251,170.375,33.529,156.311
C05166=1048.618,17.767,-77.235,170.373,33.527,156.311
C05167=1048.611,17.518,-77.220,170.371,33.525,156.311
C05168=1048.605,17.268,-77.204,170.369,33.524,156.310
C05169=1048.599,17.019,-77.189,170.368,33.522,156.310
C05170=1048.592,16.770,-77.173,170.366,33.520,156.310
C05171=1048.587,16.520,-77.158,170.364,33.518,156.310
C05172=1048.580,16.271,-77.142,170.363,33.516,156.309
C05173=1048.574,16.021,-77.126,170.361,33.515,156.309
C05174=1048.568,15.772,-77.111,170.359,33.513,156.309
C05175=1048.561,15.523,-77.095,170.357,33.512,156.309
C05176=1048.555,15.273,-77.079,170.356,33.510,156.308
C05177=1048.549,15.024,-77.064,170.354,33.508,156.308
C05178=1048.544,14.774,-77.049,170.352,33.506,156.308
C05179=1048.537,14.525,-77.034,170.350,33.504,156.307
C05180=1048.530,14.276,-77.018,170.348,33.503,156.307
C05181=1048.525,14.026,-77.002,170.346,33.501,156.307
C05182=1048.518,13.777,-76.987,170.344,33.499,156.307
C05183=1048.511,13.491,-76.969,170.342,33.497,156.306
C05184=1048.503,13.206,-76.951,170.340,33.495,156.306
C05185=1048.496,12.922,-76.934,170.338,33.493,156.306
C05186=1048.489,12.637,-76.916,170.336,33.492,156.306
C05187=1048.482,12.387,-76.902,170.334,33.490,156.305
C05188=1048.476,12.137,-76.887,170.332,33.489,156.305
C05189=1048.469,11.888,-76.871,170.331,33.487,156.305
C05190=1048.463,11.639,-76.856,170.329,33.485,156.305
C05191=1048.456,11.390,-76.840,170.327,33.483,156.304
C05192=1048.450,11.140,-76.825,170.325,33.482,156.304
C05193=1048.445,10.891,-76.810,170.324,33.480,156.304
C05194=1048.438,10.642,-76.795,170.322,33.478,156.304
C05195=1048.432,10.392,-76.780,170.320,33.477,156.303
C05196=1048.425,10.142,-76.765,170.318,33.475,156.303
C05197=1048.419,9.893,-76.749,170.317,33.474,156.303
C05198=1048.412,9.644,-76.734,170.315,33.472,156.303
C05199=1048.406,9.394,-76.718,170.313,33.470,156.302
C05200=1048.400,9.144,-76.704,170.311,33.468,156.302
C05201=1048.393,8.895,-76.688,170.309,33.467,156.302
C05202=1048.387,8.645,-76.673,170.308,33.465,156.302
C05203=1048.381,8.396,-76.658,170.306,33.463,156.301
C05204=1048.374,8.146,-76.643,170.304,33.462,156.301
C05205=1048.368,7.898,-76.628,170.302,33.460,156.301
C05206=1048.362,7.648,-76.613,170.301,33.459,156.301
C05207=1048.356,7.398,-76.597,170.299,33.457,156.300
C05208=1048.350,7.148,-76.582,170.297,33.455,156.300
C05209=1048.343,6.899,-76.567,170.295,33.453,156.300
C05210=1048.337,6.650,-76.552,170.293,33.452,156.300
C05211=1048.330,6.400,-76.537,170.292,33.450,156.299
C05212=1048.325,6.151,-76.522,170.290,33.448,156.299
C05213=1048.318,5.901,-76.507,170.288,33.447,156.299
C05214=1048.311,5.652,-76.492,170.286,33.445,156.299
C05215=1048.305,5.403,-76.477,170.285,33.444,156.298
C05216=1048.299,5.153,-76.461,170.283,33.442,156.298
C05217=1048.293,4.903,-76.446,170.281,33.440,156.298
C05218=1048.287,4.654,-76.432,170.279,33.438,156.298
C05219=1048.281,4.404,-76.417,170.277,33.437,156.297
C05220=1048.274,4.155,-76.402,170.276,33.436,156.297
C05221=1048.268,3.906,-76.386,170.274,33.433,156.297
C05222=1048.261,3.656,-76.371,170.272,33.432,156.297
C05223=1048.255,3.406,-76.356,170.270,33.430,156.296
C05224=1048.249,3.157,-76.342,170.268,33.429,156.296
C05225=1048.243,2.908,-76.327,170.267,33.427,156.296
C05226=1048.236,2.658,-76.312,170.265,33.425,156.296
C05227=1048.230,2.408,-76.297,170.263,33.424,156.296
C05228=1048.225,2.159,-76.282,170.261,33.422,156.295
C05229=1048.219,1.910,-76.267,170.259,33.420,156.295
C05230=1048.212,1.660,-76.252,170.258,33.418,156.295
C05231=1048.206,1.410,-76.237,170.256,33.417,156.295
C05232=1048.200,1.161,-76.222,170.254,33.415,156.294
C05233=1048.194,0.912,-76.207,170.252,33.414,156.294
C05234=1048.187,0.662,-76.192,170.250,33.412,156.294
C05235=1048.181,0.412,-76.177,170.249,33.410,156.294
C05236=1048.175,0.163,-76.163,170.247,33.409,156.293
C05237=1048.169,-0.086,-76.148,170.245,33.407,156.293
C05238=1048.162,-0.336,-76.133,170.243,33.405,156.293
C05239=1048.156,-0.586,-76.118,170.241,33.403,156.293
C05240=1048.150,-0.835,-76.103,170.240,33.402,156.292
C05241=1048.144,-1.084,-76.088,170.238,33.400,156.292
C05242=1048.138,-1.334,-76.073,170.236,33.399,156.292
C05243=1048.132,-1.583,-76.059,170.234,33.397,156.292
C05244=1048.125,-1.833,-76.044,170.232,33.395,156.291
C05245=1048.119,-2.082,-76.029,170.231,33.394,156.291
C05246=1048.113,-2.331,-76.014,170.229,33.392,156.291
C05247=1048.107,-2.614,-75.997,170.227,33.390,156.291
C05248=1048.099,-2.898,-75.980,170.225,33.388,156.290
C05249=1048.092,-3.181,-75.963,170.223,33.386,156.290
C05250=1048.086,-3.463,-75.947,170.221,33.384,156.290
C05251=1048.079,-3.713,-75.932,170.219,33.383,156.290
C05252=1048.073,-3.963,-75.917,170.217,33.381,156.289
C05253=1048.066,-4.212,-75.903,170.215,33.379,156.289
C05254=1048.060,-4.461,-75.888,170.213,33.378,156.289
C05255=1048.054,-4.711,-75.874,170.211,33.377,156.289
C05256=1048.047,-4.961,-75.859,170.210,33.375,156.288
C05257=1048.040,-5.210,-75.845,170.208,33.373,156.288
C05258=1048.035,-5.459,-75.830,170.206,33.372,156.288
C05259=1048.028,-5.709,-75.815,170.204,33.370,156.288
C05260=1048.022,-5.959,-75.801,170.202,33.369,156.288
C05261=1048.016,-6.208,-75.787,170.200,33.368,156.287
C05262=1048.009,-6.457,-75.772,170.199,33.366,156.287
C05263=1048.003,-6.707,-75.757,170.197,33.364,156.287
C05264=1047.997,-6.956,-75.744,170.195,33.363,156.287
C05265=1047.990,-7.206,-75.729,170.193,33.361,156.287
C05266=1047.984,-7.456,-75.714,170.191,33.359,156.286
C05267=1047.978,-7.705,-75.700,170.189,33.358,156.286
C05268=1047.971,-7.955,-75.686,170.187,33.357,156.286
C05269=1047.965,-8.204,-75.671,170.186,33.355,156.286
C05270=1047.959,-8.453,-75.656,170.184,33.353,156.285
C05271=1047.953,-8.704,-75.642,170.182,33.352,156.285
C05272=1047.946,-8.953,-75.628,170.180,33.350,156.285
C05273=1047.940,-9.202,-75.613,170.178,33.349,156.285
C05274=1047.934,-9.452,-75.599,170.176,33.347,156.284
C05275=1047.927,-9.701,-75.585,170.174,33.345,156.284
C05276=1047.921,-9.950,-75.570,170.173,33.344,156.284
C05277=1047.915,-10.201,-75.556,170.171,33.343,156.284
C05278=1047.909,-10.449,-75.542,170.169,33.341,156.284
C05279=1047.902,-10.700,-75.528,170.167,33.339,156.283
C05280=1047.897,-10.949,-75.513,170.165,33.338,156.283
C05281=1047.890,-11.198,-75.499,170.163,33.336,156.283
C05282=1047.883,-11.448,-75.484,170.161,33.335,156.283
C05283=1047.878,-11.697,-75.470,170.160,33.333,156.282
C05284=1047.872,-11.947,-75.456,170.158,33.332,156.282
C05285=1047.865,-12.196,-75.442,170.156,33.330,156.282
C05286=1047.859,-12.446,-75.427,170.154,33.329,156.282
C05287=1047.853,-12.695,-75.413,170.152,33.327,156.282
C05288=1047.846,-12.945,-75.398,170.150,33.325,156.281
C05289=1047.840,-13.195,-75.384,170.148,33.324,156.281
C05290=1047.834,-13.444,-75.370,170.146,33.322,156.281
C05291=1047.827,-13.694,-75.356,170.145,33.321,156.281
C05292=1047.822,-13.943,-75.341,170.143,33.319,156.281
C05293=1047.816,-14.193,-75.327,170.141,33.318,156.280
C05294=1047.809,-14.442,-75.313,170.139,33.316,156.280
C05295=1047.803,-14.692,-75.299,170.137,33.315,156.280
C05296=1047.797,-14.941,-75.284,170.135,33.313,156.280
C05297=1047.790,-15.191,-75.271,170.133,33.311,156.279
C05298=1047.785,-15.440,-75.256,170.132,33.310,156.279
C05299=1047.778,-15.690,-75.243,170.130,33.309,156.279
C05300=1047.771,-15.939,-75.228,170.129,33.307,156.279
C05301=1047.765,-16.189,-75.214,170.127,33.306,156.279
C05302=1047.758,-16.439,-75.201,170.125,33.304,156.279
C05303=1047.753,-16.688,-75.186,170.123,33.303,156.278
C05304=1047.746,-16.938,-75.173,170.121,33.302,156.278
C05305=1047.740,-17.187,-75.158,170.119,33.300,156.278
C05306=1047.733,-17.437,-75.144,170.117,33.299,156.278
C05307=1047.728,-17.686,-75.130,170.115,33.297,156.278
C05308=1047.721,-17.935,-75.116,170.113,33.295,156.277
C05309=1047.715,-18.185,-75.102,170.111,33.294,156.277
C05310=1047.708,-18.435,-75.089,170.110,33.292,156.277
C05311=1047.701,-18.716,-75.073,170.107,33.291,156.277
C05312=1047.694,-18.997,-75.057,170.105,33.290,156.277
C05313=1047.687,-19.279,-75.041,170.103,33.287,156.276
C05314=1047.680,-19.560,-75.025,170.101,33.286,156.276
C05315=1047.673,-19.810,-75.012,170.099,33.285,156.276
C05316=1047.668,-20.060,-74.998,170.097,33.283,156.276
C05317=1047.661,-20.308,-74.984,170.095,33.282,156.275
C05318=1047.654,-20.558,-74.970,170.093,33.280,156.275
C05319=1047.649,-20.808,-74.956,170.091,33.279,156.275
C05320=1047.642,-21.057,-74.942,170.089,33.278,156.275
C05321=1047.636,-21.307,-74.928,170.087,33.276,156.275
C05322=1047.629,-21.557,-74.914,170.086,33.275,156.275
C05323=1047.623,-21.806,-74.901,170.084,33.273,156.274
C05324=1047.617,-22.056,-74.886,170.082,33.272,156.274
C05325=1047.611,-22.305,-74.873,170.080,33.270,156.274
C05326=1047.605,-22.555,-74.859,170.078,33.268,156.274
C05327=1047.598,-22.804,-74.845,170.076,33.267,156.273
C05328=1047.592,-23.054,-74.832,170.074,33.266,156.273
C05329=1047.586,-23.303,-74.817,170.072,33.264,156.273
C05330=1047.580,-23.553,-74.804,170.070,33.263,156.273
C05331=1047.573,-23.802,-74.791,170.068,33.261,156.273
C05332=1047.567,-24.052,-74.776,170.066,33.260,156.273
C05333=1047.561,-24.301,-74.763,170.064,33.258,156.272
C05334=1047.555,-24.552,-74.749,170.062,33.257,156.272
C05335=1047.548,-24.800,-74.735,170.061,33.256,156.272
C05336=1047.542,-25.050,-74.722,170.059,33.254,156.272
C05337=1047.536,-25.300,-74.707,170.057,33.253,156.272
C05338=1047.530,-25.549,-74.694,170.055,33.251,156.271
C05339=1047.524,-25.798,-74.681,170.053,33.250,156.271
C05340=1047.518,-26.049,-74.667,170.051,33.249,156.271
C05341=1047.511,-26.298,-74.653,170.049,33.247,156.271
C05342=1047.506,-26.548,-74.640,170.047,33.246,156.271
C05343=1047.499,-26.798,-74.626,170.045,33.244,156.270
C05344=1047.493,-27.047,-74.613,170.043,33.243,156.270
C05345=1047.486,-27.295,-74.599,170.041,33.241,156.270
C05346=1047.480,-27.545,-74.585,170.039,33.240,156.270
C05347=1047.474,-27.795,-74.571,170.037,33.239,156.270
C05348=1047.467,-28.045,-74.558,170.035,33.237,156.270
C05349=1047.461,-28.294,-74.544,170.033,33.236,156.269
C05350=1047.455,-28.543,-74.531,170.031,33.235,156.269
C05351=1047.448,-28.793,-74.517,170.029,33.234,156.269
C05352=1047.442,-29.043,-74.504,170.027,33.232,156.269
C05353=1047.436,-29.292,-74.491,170.025,33.231,156.269
C05354=1047.429,-29.543,-74.478,170.023,33.229,156.269
C05355=1047.424,-29.792,-74.464,170.021,33.228,156.268
C05356=1047.417,-30.041,-74.451,170.019,33.227,156.268
C05357=1047.411,-30.291,-74.437,170.017,33.226,156.268
C05358=1047.404,-30.541,-74.424,170.015,33.224,156.268
C05359=1047.398,-30.790,-74.411,170.014,33.223,156.268
C05360=1047.391,-31.040,-74.397,170.012,33.221,156.267
C05361=1047.385,-31.289,-74.384,170.010,33.220,156.267
C05362=1047.379,-31.538,-74.370,170.008,33.219,156.267
C05363=1047.373,-31.788,-74.357,170.006,33.218,156.267
C05364=1047.367,-32.038,-74.343,170.004,33.216,156.267
C05365=1047.360,-32.287,-74.330,170.002,33.215,156.267
C05366=1047.355,-32.537,-74.317,170.000,33.213,156.266
C05367=1047.348,-32.787,-74.303,169.998,33.212,156.266
C05368=1047.341,-33.036,-74.290,169.996,33.211,156.266
C05369=1047.335,-33.286,-74.277,169.994,33.209,156.266
C05370=1047.329,-33.535,-74.264,169.992,33.208,156.266
C05371=1047.322,-33.785,-74.250,169.990,33.207,156.266
C05372=1047.316,-34.035,-74.237,169.989,33.205,156.265
C05373=1047.310,-34.284,-74.224,169.987,33.204,156.265
C05374=1047.304,-34.533,-74.211,169.985,33.203,156.265
C05375=1047.297,-34.814,-74.195,169.983,33.201,156.265
C05376=1047.290,-35.094,-74.180,169.980,33.200,156.265
C05377=1047.283,-35.375,-74.166,169.978,33.198,156.265
C05378=1047.276,-35.656,-74.151,169.976,33.197,156.264
C05379=1047.270,-35.905,-74.137,169.974,33.195,156.264
C05380=1047.264,-36.155,-74.125,169.972,33.195,156.264
C05381=1047.258,-36.405,-74.112,169.970,33.193,156.264
C05382=1047.251,-36.655,-74.098,169.968,33.192,156.264
C05383=1047.245,-36.904,-74.085,169.966,33.190,156.264
C05384=1047.239,-37.154,-74.072,169.964,33.189,156.263
C05385=1047.233,-37.403,-74.059,169.962,33.187,156.263
C05386=1047.227,-37.652,-74.046,169.960,33.187,156.263
C05387=1047.220,-37.902,-74.032,169.958,33.185,156.263
C05388=1047.214,-38.152,-74.019,169.956,33.184,156.263
C05389=1047.208,-38.401,-74.006,169.954,33.182,156.263
C05390=1047.201,-38.651,-73.993,169.952,33.181,156.262
C05391=1047.195,-38.901,-73.980,169.950,33.180,156.262
C05392=1047.189,-39.150,-73.967,169.948,33.179,156.262
C05393=1047.183,-39.400,-73.954,169.946,33.177,156.262
C05394=1047.177,-39.650,-73.941,169.944,33.176,156.262
C05395=1047.170,-39.899,-73.928,169.942,33.175,156.262
C05396=1047.164,-40.148,-73.916,169.940,33.174,156.262
C05397=1047.157,-40.398,-73.902,169.938,33.173,156.261
C05398=1047.152,-40.648,-73.890,169.936,33.171,156.261
C05399=1047.145,-40.898,-73.876,169.934,33.171,156.261
C05400=1047.139,-41.147,-73.863,169.931,33.169,156.261
C05401=1047.132,-41.396,-73.851,169.929,33.168,156.261
C05402=1047.126,-41.646,-73.838,169.927,33.167,156.261
C05403=1047.120,-41.896,-73.825,169.925,33.165,156.261
C05404=1047.114,-42.145,-73.812,169.923,33.164,156.260
C05405=1047.108,-42.395,-73.799,169.921,33.163,156.260
C05406=1047.100,-42.644,-73.786,169.919,33.162,156.260
C05407=1047.094,-42.894,-73.774,169.917,33.161,156.260
C05408=1047.088,-43.144,-73.760,169.915,33.159,156.260
C05409=1047.082,-43.393,-73.748,169.913,33.158,156.260
C05410=1047.076,-43.643,-73.735,169.911,33.157,156.260
C05411=1047.069,-43.892,-73.723,169.909,33.156,156.259
C05412=1047.063,-44.141,-73.709,169.907,33.154,156.259
C05413=1047.057,-44.391,-73.697,169.905,33.153,156.259
C05414=1047.051,-44.641,-73.683,169.903,33.152,156.259
C05415=1047.045,-44.891,-73.671,169.901,33.151,156.259
C05416=1047.038,-45.140,-73.659,169.899,33.150,156.259
C05417=1047.032,-45.389,-73.646,169.897,33.148,156.259
C05418=1047.026,-45.640,-73.633,169.895,33.148,156.258
C05419=1047.019,-45.889,-73.619,169.893,33.146,156.258
C05420=1047.013,-46.139,-73.608,169.892,33.145,156.258
C05421=1047.007,-46.389,-73.595,169.890,33.144,156.258
C05422=1047.001,-46.638,-73.582,169.887,33.143,156.258
C05423=1046.995,-46.888,-73.569,169.885,33.142,156.258
C05424=1046.988,-47.137,-73.556,169.883,33.140,156.258
C05425=1046.982,-47.387,-73.544,169.881,33.139,156.258
C05426=1046.976,-47.637,-73.531,169.879,33.138,156.257
C05427=1046.970,-47.886,-73.518,169.877,33.137,156.257
C05428=1046.964,-48.136,-73.506,169.875,33.136,156.257
C05429=1046.957,-48.385,-73.494,169.873,33.134,156.257
C05430=1046.951,-48.635,-73.480,169.871,33.133,156.257
C05431=1046.945,-48.884,-73.468,169.869,33.132,156.257
C05432=1046.939,-49.134,-73.455,169.867,33.131,156.257
C05433=1046.932,-49.383,-73.443,169.865,33.130,156.256
C05434=1046.926,-49.633,-73.430,169.863,33.129,156.256
C05435=1046.920,-49.883,-73.417,169.861,33.127,156.256
C05436=1046.914,-50.133,-73.405,169.859,33.127,156.256
C05437=1046.907,-50.382,-73.392,169.857,33.125,156.256
C05438=1046.902,-50.632,-73.380,169.854,33.124,156.256
C05439=1046.895,-50.912,-73.366,169.852,33.123,156.256
C05440=1046.887,-51.194,-73.352,169.850,33.122,156.256
C05441=1046.880,-51.475,-73.338,169.847,33.120,156.255
